LIN {X 0,Y 509.374,Z 538.173,A -85,B 0,C 180,E1 19045.4,E2 19045.4} C_VEL
LIN {X 0,Y 505.626,Z 523.597,A -85,B 0,C 180,E1 19044.365,E2 19044.365} C_VEL
LIN {X 0,Y 504.714,Z 520.545,A -85,B 0,C 180,E1 19044.099,E2 19044.099} C_VEL
LIN {X 0,Y 504.683,Z 520.186,A -85,B 0,C 180,E1 19043.675,E2 19043.675} C_VEL
LIN {X 0,Y 504.675,Z 520.134,A -85,B 0,C 180,E1 19040.214,E2 19040.214} C_VEL
LIN {X 0,Y 504.748,Z 520.47,A -85,B 0,C 180,E1 19039.175,E2 19039.175} C_VEL
LIN {X 0,Y 506.259,Z 524.019,A -85,B 0,C 180,E1 19038.577,E2 19038.577} C_VEL
LIN {X 0,Y 514.07,Z 540.46,A -85,B 0,C 180,E1 19036.024,E2 19036.024} C_VEL
LIN {X 0,Y 516.619,Z 546.048,A -85,B 0,C 180,E1 19035.262,E2 19035.262} C_VEL
LIN {X 0,Y 526.038,Z 560.599,A -85,B 0,C 180,E1 19034.052,E2 19034.052} C_VEL
LIN {X 0,Y 527.632,Z 568.688,A -85,B 0,C 180,E1 19033.753,E2 19033.753} C_VEL
LIN {X 0,Y 524.708,Z 775.867,A -85,B 0,C 180,E1 19030.439,E2 19030.439} C_VEL
LIN {X 0,Y 522.743,Z 892.473,A -85,B 0,C 180,E1 19028.548,E2 19028.548} C_VEL
LIN {X 0,Y 521.824,Z 915.213,A -85,B 0,C 180,E1 19027.996,E2 19027.996} C_VEL
LIN {X 0,Y 520.789,Z 935.158,A -85,B 0,C 180,E1 19027.346,E2 19027.346} C_VEL
LIN {X 0,Y 519.279,Z 958.378,A -85,B 0,C 180,E1 19026.374,E2 19026.374} C_VEL
LIN {X 0,Y 517.768,Z 979.695,A -85,B 0,C 180,E1 19025.268,E2 19025.268} C_VEL
LIN {X 0,Y 516.05,Z 1000.225,A -85,B 0,C 180,E1 19023.978,E2 19023.978} C_VEL
LIN {X 0,Y 514.336,Z 1020.252,A -85,B 0,C 180,E1 19022.508,E2 19022.508} C_VEL
LIN {X 0,Y 512.59,Z 1039.264,A -85,B 0,C 180,E1 19020.865,E2 19020.865} C_VEL
LIN {X 0,Y 510.801,Z 1058.785,A -85,B 0,C 180,E1 19018.914,E2 19018.914} C_VEL
LIN {X 0,Y 509.332,Z 1075.15,A -85,B 0,C 180,E1 19017.03,E2 19017.03} C_VEL
LIN {X 0,Y 507.958,Z 1091.142,A -85,B 0,C 180,E1 19014.913,E2 19014.913} C_VEL
LIN {X 0,Y 506.773,Z 1106.221,A -85,B 0,C 180,E1 19012.627,E2 19012.627} C_VEL
LIN {X 0,Y 505.853,Z 1119.088,A -85,B 0,C 180,E1 19010.358,E2 19010.358} C_VEL
LIN {X 0,Y 505.083,Z 1131.807,A -85,B 0,C 180,E1 19007.75,E2 19007.75} C_VEL
LIN {X 0,Y 504.598,Z 1141.528,A -85,B 0,C 180,E1 19005.398,E2 19005.398} C_VEL
LIN {X 0,Y 504.238,Z 1150.346,A -85,B 0,C 180,E1 19002.832,E2 19002.832} C_VEL
LIN {X 0,Y 504.07,Z 1156.866,A -85,B 0,C 180,E1 19000.515,E2 19000.515} C_VEL
LIN {X 0,Y 503.966,Z 1162.635,A -85,B 0,C 180,E1 18997.868,E2 18997.868} C_VEL
LIN {X 0,Y 503.904,Z 1166.278,A -85,B 0,C 180,E1 18995.58,E2 18995.58} C_VEL
LIN {X 0,Y 503.889,Z 1168.919,A -85,B 0,C 180,E1 18992.957,E2 18992.957} C_VEL
LIN {X 0,Y 503.884,Z 1169.872,A -85,B 0,C 180,E1 18990.682,E2 18990.682} C_VEL
LIN {X 0,Y 503.907,Z 1169.526,A -85,B 0,C 180,E1 18988.067,E2 18988.067} C_VEL
LIN {X 0,Y 503.913,Z 1167.729,A -85,B 0,C 180,E1 18985.676,E2 18985.676} C_VEL
LIN {X 0,Y 503.923,Z 1164.494,A -85,B 0,C 180,E1 18983.163,E2 18983.163} C_VEL
LIN {X 0,Y 504.003,Z 1159.828,A -85,B 0,C 180,E1 18980.753,E2 18980.753} C_VEL
LIN {X 0,Y 504.156,Z 1153.517,A -85,B 0,C 180,E1 18978.213,E2 18978.213} C_VEL
LIN {X 0,Y 504.423,Z 1145.344,A -85,B 0,C 180,E1 18975.654,E2 18975.654} C_VEL
LIN {X 0,Y 504.885,Z 1135.421,A -85,B 0,C 180,E1 18973.075,E2 18973.075} C_VEL
LIN {X 0,Y 505.497,Z 1124.573,A -85,B 0,C 180,E1 18970.712,E2 18970.712} C_VEL
LIN {X 0,Y 506.398,Z 1111.156,A -85,B 0,C 180,E1 18968.21,E2 18968.21} C_VEL
LIN {X 0,Y 507.492,Z 1097.01,A -85,B 0,C 180,E1 18965.931,E2 18965.931} C_VEL
LIN {X 0,Y 508.795,Z 1081.335,A -85,B 0,C 180,E1 18963.758,E2 18963.758} C_VEL
LIN {X 0,Y 510.309,Z 1064.33,A -85,B 0,C 180,E1 18961.696,E2 18961.696} C_VEL
LIN {X 0,Y 511.832,Z 1047.548,A -85,B 0,C 180,E1 18959.927,E2 18959.927} C_VEL
LIN {X 0,Y 513.655,Z 1027.52,A -85,B 0,C 180,E1 18958.096,E2 18958.096} C_VEL
LIN {X 0,Y 515.411,Z 1008.083,A -85,B 0,C 180,E1 18956.568,E2 18956.568} C_VEL
LIN {X 0,Y 517.065,Z 987.821,A -85,B 0,C 180,E1 18955.218,E2 18955.218} C_VEL
LIN {X 0,Y 518.718,Z 967.181,A -85,B 0,C 180,E1 18954.054,E2 18954.054} C_VEL
LIN {X 0,Y 520.087,Z 946.602,A -85,B 0,C 180,E1 18953.106,E2 18953.106} C_VEL
LIN {X 0,Y 521.311,Z 925.729,A -85,B 0,C 180,E1 18952.321,E2 18952.321} C_VEL
LIN {X 0,Y 522.324,Z 902.992,A -85,B 0,C 180,E1 18951.682,E2 18951.682} C_VEL
LIN {X 0,Y 523.077,Z 879.403,A -85,B 0,C 180,E1 18951.217,E2 18951.217} C_VEL
LIN {X 0,Y 525.528,Z 712.407,A -85,B 0,C 180,E1 18948.56,E2 18948.56} C_VEL
LIN {X 0,Y 527.601,Z 563.686,A -85,B 0,C 180,E1 18946.153,E2 18946.153} C_VEL
LIN {X 0,Y 526.674,Z 559.647,A -85,B 0,C 180,E1 18945.992,E2 18945.992} C_VEL
LIN {X 0,Y 516.407,Z 544.042,A -85,B 0,C 180,E1 18944.654,E2 18944.654} C_VEL
LIN {X 0,Y 508.668,Z 528.582,A -85,B 0,C 180,E1 18942.545,E2 18942.545} C_VEL
LIN {X 0,Y 506.242,Z 523.996,A -85,B 0,C 180,E1 18941.875,E2 18941.875} C_VEL
LIN {X 0,Y 504.741,Z 520.388,A -85,B 0,C 180,E1 18941.325,E2 18941.325} C_VEL
LIN {X 0,Y 504.697,Z 520.161,A -85,B 0,C 180,E1 18937.771,E2 18937.771} C_VEL
LIN {X 0,Y 504.694,Z 520.181,A -85,B 0,C 180,E1 18934.238,E2 18934.238} C_VEL
LIN {X 0,Y 504.711,Z 520.174,A -85,B 0,C 180,E1 18930.708,E2 18930.708} C_VEL
LIN {X 0,Y 504.695,Z 520.153,A -85,B 0,C 180,E1 18927.186,E2 18927.186} C_VEL
LIN {X 0,Y 504.695,Z 520.179,A -85,B 0,C 180,E1 18923.713,E2 18923.713} C_VEL
LIN {X 0,Y 504.703,Z 520.168,A -85,B 0,C 180,E1 18920.164,E2 18920.164} C_VEL
LIN {X 0,Y 504.697,Z 520.159,A -85,B 0,C 180,E1 18916.694,E2 18916.694} C_VEL
LIN {X 0,Y 504.694,Z 520.17,A -85,B 0,C 180,E1 18913.169,E2 18913.169} C_VEL
LIN {X 0,Y 504.699,Z 520.157,A -85,B 0,C 180,E1 18909.694,E2 18909.694} C_VEL
LIN {X 0,Y 504.697,Z 520.176,A -85,B 0,C 180,E1 18906.141,E2 18906.141} C_VEL
LIN {X 0,Y 504.695,Z 520.173,A -85,B 0,C 180,E1 18902.611,E2 18902.611} C_VEL
LIN {X 0,Y 504.702,Z 520.173,A -85,B 0,C 180,E1 18899.092,E2 18899.092} C_VEL
LIN {X 0,Y 504.695,Z 520.178,A -85,B 0,C 180,E1 18895.568,E2 18895.568} C_VEL
LIN {X 0,Y 504.698,Z 520.171,A -85,B 0,C 180,E1 18892.119,E2 18892.119} C_VEL
LIN {X 0,Y 504.695,Z 520.16,A -85,B 0,C 180,E1 18888.573,E2 18888.573} C_VEL
LIN {X 0,Y 504.693,Z 520.179,A -85,B 0,C 180,E1 18884.958,E2 18884.958} C_VEL
LIN {X 0,Y 504.698,Z 520.155,A -85,B 0,C 180,E1 18881.52,E2 18881.52} C_VEL
LIN {X 0,Y 504.698,Z 520.177,A -85,B 0,C 180,E1 18877.996,E2 18877.996} C_VEL
LIN {X 0,Y 504.69,Z 520.153,A -85,B 0,C 180,E1 18874.412,E2 18874.412} C_VEL
LIN {X 0,Y 504.701,Z 520.175,A -85,B 0,C 180,E1 18870.887,E2 18870.887} C_VEL
LIN {X 0,Y 504.7,Z 520.176,A -85,B 0,C 180,E1 18867.349,E2 18867.349} C_VEL
LIN {X 0,Y 504.685,Z 520.158,A -85,B 0,C 180,E1 18863.739,E2 18863.739} C_VEL
LIN {X 0,Y 504.699,Z 520.158,A -85,B 0,C 180,E1 18860.363,E2 18860.363} C_VEL
LIN {X 0,Y 504.689,Z 520.163,A -85,B 0,C 180,E1 18856.883,E2 18856.883} C_VEL
LIN {X 0,Y 504.772,Z 520.605,A -85,B 0,C 180,E1 18856.246,E2 18856.246} C_VEL
LIN {X 0,Y 506.506,Z 524.334,A -85,B 0,C 180,E1 18855.668,E2 18855.668} C_VEL
LIN {X 0,Y 515.146,Z 542.071,A -85,B 0,C 180,E1 18853.131,E2 18853.131} C_VEL
LIN {X 0,Y 516.768,Z 545.52,A -85,B 0,C 180,E1 18852.666,E2 18852.666} C_VEL
LIN {X 0,Y 517.661,Z 549.436,A -85,B 0,C 180,E1 18852.245,E2 18852.245} C_VEL
LIN {X 0,Y 517.414,Z 555.801,A -85,B 0,C 180,E1 18851.744,E2 18851.744} C_VEL
LIN {X 0,Y 513.944,Z 574.599,A -85,B 0,C 180,E1 18850.556,E2 18850.556} C_VEL
LIN {X 0,Y 513.868,Z 575.564,A -85,B 0,C 180,E1 18850.486,E2 18850.486} C_VEL
LIN {X 0,Y 513.159,Z 588.697,A -85,B 0,C 180,E1 18849.537,E2 18849.537} C_VEL
LIN {X 0,Y 516.897,Z 611.864,A -85,B 0,C 180,E1 18848.752,E2 18848.752} C_VEL
LIN {X 0,Y 513.011,Z 833.068,A -85,B 0,C 180,E1 18845.203,E2 18845.203} C_VEL
LIN {X 0,Y 511.794,Z 896.976,A -85,B 0,C 180,E1 18844.15,E2 18844.15} C_VEL
LIN {X 0,Y 510.861,Z 917.747,A -85,B 0,C 180,E1 18843.613,E2 18843.613} C_VEL
LIN {X 0,Y 509.667,Z 940.451,A -85,B 0,C 180,E1 18842.816,E2 18842.816} C_VEL
LIN {X 0,Y 508.463,Z 960.06,A -85,B 0,C 180,E1 18841.936,E2 18841.936} C_VEL
LIN {X 0,Y 506.93,Z 980.559,A -85,B 0,C 180,E1 18840.786,E2 18840.786} C_VEL
LIN {X 0,Y 505.393,Z 1000.249,A -85,B 0,C 180,E1 18839.448,E2 18839.448} C_VEL
LIN {X 0,Y 503.85,Z 1018.516,A -85,B 0,C 180,E1 18837.984,E2 18837.984} C_VEL
LIN {X 0,Y 502.296,Z 1036.377,A -85,B 0,C 180,E1 18836.289,E2 18836.289} C_VEL
LIN {X 0,Y 500.843,Z 1052.997,A -85,B 0,C 180,E1 18834.448,E2 18834.448} C_VEL
LIN {X 0,Y 499.563,Z 1068.367,A -85,B 0,C 180,E1 18832.475,E2 18832.475} C_VEL
LIN {X 0,Y 498.455,Z 1082.852,A -85,B 0,C 180,E1 18830.305,E2 18830.305} C_VEL
LIN {X 0,Y 497.584,Z 1095.279,A -85,B 0,C 180,E1 18828.11,E2 18828.11} C_VEL
LIN {X 0,Y 496.885,Z 1107.121,A -85,B 0,C 180,E1 18825.643,E2 18825.643} C_VEL
LIN {X 0,Y 496.443,Z 1116.603,A -85,B 0,C 180,E1 18823.274,E2 18823.274} C_VEL
LIN {X 0,Y 496.165,Z 1124.245,A -85,B 0,C 180,E1 18820.919,E2 18820.919} C_VEL
LIN {X 0,Y 496.006,Z 1130.548,A -85,B 0,C 180,E1 18818.462,E2 18818.462} C_VEL
LIN {X 0,Y 495.933,Z 1135.255,A -85,B 0,C 180,E1 18816.018,E2 18816.018} C_VEL
LIN {X 0,Y 495.907,Z 1138.243,A -85,B 0,C 180,E1 18813.583,E2 18813.583} C_VEL
LIN {X 0,Y 495.908,Z 1139.793,A -85,B 0,C 180,E1 18811.04,E2 18811.04} C_VEL
LIN {X 0,Y 495.908,Z 1139.767,A -85,B 0,C 180,E1 18808.729,E2 18808.729} C_VEL
LIN {X 0,Y 495.907,Z 1138.105,A -85,B 0,C 180,E1 18806.185,E2 18806.185} C_VEL
LIN {X 0,Y 495.941,Z 1134.893,A -85,B 0,C 180,E1 18803.685,E2 18803.685} C_VEL
LIN {X 0,Y 496.014,Z 1130.234,A -85,B 0,C 180,E1 18801.304,E2 18801.304} C_VEL
LIN {X 0,Y 496.175,Z 1123.81,A -85,B 0,C 180,E1 18798.846,E2 18798.846} C_VEL
LIN {X 0,Y 496.469,Z 1116.095,A -85,B 0,C 180,E1 18796.49,E2 18796.49} C_VEL
LIN {X 0,Y 496.927,Z 1106.429,A -85,B 0,C 180,E1 18794.108,E2 18794.108} C_VEL
LIN {X 0,Y 497.605,Z 1094.92,A -85,B 0,C 180,E1 18791.732,E2 18791.732} C_VEL
LIN {X 0,Y 498.501,Z 1082.19,A -85,B 0,C 180,E1 18789.501,E2 18789.501} C_VEL
LIN {X 0,Y 499.582,Z 1068.129,A -85,B 0,C 180,E1 18787.402,E2 18787.402} C_VEL
LIN {X 0,Y 500.879,Z 1052.572,A -85,B 0,C 180,E1 18785.411,E2 18785.411} C_VEL
LIN {X 0,Y 502.377,Z 1035.417,A -85,B 0,C 180,E1 18783.524,E2 18783.524} C_VEL
LIN {X 0,Y 503.893,Z 1018.046,A -85,B 0,C 180,E1 18781.883,E2 18781.883} C_VEL
LIN {X 0,Y 505.437,Z 999.747,A -85,B 0,C 180,E1 18780.425,E2 18780.425} C_VEL
LIN {X 0,Y 506.985,Z 979.853,A -85,B 0,C 180,E1 18779.081,E2 18779.081} C_VEL
LIN {X 0,Y 508.446,Z 960.379,A -85,B 0,C 180,E1 18777.99,E2 18777.99} C_VEL
LIN {X 0,Y 509.681,Z 940.217,A -85,B 0,C 180,E1 18777.084,E2 18777.084} C_VEL
LIN {X 0,Y 510.897,Z 917.075,A -85,B 0,C 180,E1 18776.277,E2 18776.277} C_VEL
LIN {X 0,Y 511.811,Z 896.306,A -85,B 0,C 180,E1 18775.746,E2 18775.746} C_VEL
LIN {X 0,Y 513.921,Z 783.082,A -85,B 0,C 180,E1 18773.904,E2 18773.904} C_VEL
LIN {X 0,Y 516.736,Z 613.605,A -85,B 0,C 180,E1 18771.173,E2 18771.173} C_VEL
LIN {X 0,Y 511.613,Z 588.579,A -85,B 0,C 180,E1 18770.179,E2 18770.179} C_VEL
LIN {X 0,Y 513.574,Z 559.712,A -85,B 0,C 180,E1 18767.55,E2 18767.55} C_VEL
LIN {X 0,Y 507.022,Z 544.118,A -85,B 0,C 180,E1 18765.229,E2 18765.229} C_VEL
LIN {X 0,Y 500.324,Z 529.196,A -85,B 0,C 180,E1 18762.802,E2 18762.802} C_VEL
LIN {X 0,Y 496.818,Z 521.605,A -85,B 0,C 180,E1 18761.462,E2 18761.462} C_VEL
LIN {X 0,Y 496.742,Z 521.125,A -85,B 0,C 180,E1 18760.814,E2 18760.814} C_VEL
LIN {X 0,Y 496.756,Z 521.438,A -85,B 0,C 180,E1 18758.385,E2 18758.385} C_VEL
LIN {X 0,Y 504.618,Z 543.801,A -85,B 0,C 180,E1 18755.961,E2 18755.961} C_VEL
LIN {X 0,Y 505.837,Z 548.641,A -85,B 0,C 180,E1 18755.474,E2 18755.474} C_VEL
LIN {X 0,Y 504.883,Z 590.98,A -85,B 0,C 180,E1 18752.048,E2 18752.048} C_VEL
LIN {X 0,Y 503.801,Z 630.683,A -85,B 0,C 180,E1 18748.834,E2 18748.834} C_VEL
LIN {X 0,Y 502.476,Z 673.939,A -85,B 0,C 180,E1 18745.33,E2 18745.33} C_VEL
LIN {X 0,Y 501.367,Z 709.763,A -85,B 0,C 180,E1 18742.454,E2 18742.454} C_VEL
LIN {X 0,Y 502.49,Z 720.165,A -85,B 0,C 180,E1 18742.24,E2 18742.24} C_VEL
LIN {X 0,Y 501.055,Z 879.658,A -85,B 0,C 180,E1 18739.834,E2 18739.834} C_VEL
LIN {X 0,Y 500.731,Z 897.059,A -85,B 0,C 180,E1 18739.361,E2 18739.361} C_VEL
LIN {X 0,Y 500.263,Z 913.355,A -85,B 0,C 180,E1 18738.705,E2 18738.705} C_VEL
LIN {X 0,Y 499.681,Z 929.581,A -85,B 0,C 180,E1 18737.828,E2 18737.828} C_VEL
LIN {X 0,Y 499.025,Z 944.8,A -85,B 0,C 180,E1 18736.77,E2 18736.77} C_VEL
LIN {X 0,Y 498.371,Z 958.85,A -85,B 0,C 180,E1 18735.536,E2 18735.536} C_VEL
LIN {X 0,Y 497.722,Z 971.827,A -85,B 0,C 180,E1 18734.128,E2 18734.128} C_VEL
LIN {X 0,Y 497.144,Z 983.648,A -85,B 0,C 180,E1 18732.546,E2 18732.546} C_VEL
LIN {X 0,Y 496.667,Z 994.101,A -85,B 0,C 180,E1 18730.791,E2 18730.791} C_VEL
LIN {X 0,Y 496.318,Z 1002.856,A -85,B 0,C 180,E1 18728.924,E2 18728.924} C_VEL
LIN {X 0,Y 496.099,Z 1009.578,A -85,B 0,C 180,E1 18727.062,E2 18727.062} C_VEL
LIN {X 0,Y 495.978,Z 1014.779,A -85,B 0,C 180,E1 18725.089,E2 18725.089} C_VEL
LIN {X 0,Y 495.929,Z 1018.358,A -85,B 0,C 180,E1 18723.005,E2 18723.005} C_VEL
LIN {X 0,Y 495.92,Z 1020.068,A -85,B 0,C 180,E1 18720.924,E2 18720.924} C_VEL
LIN {X 0,Y 495.924,Z 1020.017,A -85,B 0,C 180,E1 18718.845,E2 18718.845} C_VEL
LIN {X 0,Y 495.933,Z 1018.218,A -85,B 0,C 180,E1 18716.764,E2 18716.764} C_VEL
LIN {X 0,Y 495.996,Z 1014.584,A -85,B 0,C 180,E1 18714.68,E2 18714.68} C_VEL
LIN {X 0,Y 496.133,Z 1009.313,A -85,B 0,C 180,E1 18712.706,E2 18712.706} C_VEL
LIN {X 0,Y 496.402,Z 1002.018,A -85,B 0,C 180,E1 18710.727,E2 18710.727} C_VEL
LIN {X 0,Y 496.756,Z 993.678,A -85,B 0,C 180,E1 18708.977,E2 18708.977} C_VEL
LIN {X 0,Y 497.217,Z 983.868,A -85,B 0,C 180,E1 18707.339,E2 18707.339} C_VEL
LIN {X 0,Y 497.788,Z 972.555,A -85,B 0,C 180,E1 18705.816,E2 18705.816} C_VEL
LIN {X 0,Y 498.431,Z 959.663,A -85,B 0,C 180,E1 18704.407,E2 18704.407} C_VEL
LIN {X 0,Y 499.06,Z 945.596,A -85,B 0,C 180,E1 18703.172,E2 18703.172} C_VEL
LIN {X 0,Y 499.651,Z 931.225,A -85,B 0,C 180,E1 18702.172,E2 18702.172} C_VEL
LIN {X 0,Y 500.187,Z 914.88,A -85,B 0,C 180,E1 18701.287,E2 18701.287} C_VEL
LIN {X 0,Y 500.618,Z 898.01,A -85,B 0,C 180,E1 18700.615,E2 18700.615} C_VEL
LIN {X 0,Y 500.878,Z 880.613,A -85,B 0,C 180,E1 18700.159,E2 18700.159} C_VEL
LIN {X 0,Y 502.04,Z 716.903,A -85,B 0,C 180,E1 18697.709,E2 18697.709} C_VEL
LIN {X 0,Y 501.572,Z 712.774,A -85,B 0,C 180,E1 18697.589,E2 18697.589} C_VEL
LIN {X 0,Y 502.647,Z 670.001,A -85,B 0,C 180,E1 18694.238,E2 18694.238} C_VEL
LIN {X 0,Y 503.155,Z 631.96,A -85,B 0,C 180,E1 18691.386,E2 18691.386} C_VEL
LIN {X 0,Y 503.12,Z 597.05,A -85,B 0,C 180,E1 18688.889,E2 18688.889} C_VEL
LIN {X 0,Y 502.621,Z 562.387,A -85,B 0,C 180,E1 18686.563,E2 18686.563} C_VEL
LIN {X 0,Y 501.893,Z 540.312,A -85,B 0,C 180,E1 18685.163,E2 18685.163} C_VEL
LIN {X 0,Y 498.305,Z 526.321,A -85,B 0,C 180,E1 18684.158,E2 18684.158} C_VEL
LIN {X 0,Y 496.798,Z 521.567,A -85,B 0,C 180,E1 18683.756,E2 18683.756} C_VEL
LIN {X 0,Y 496.763,Z 521.172,A -85,B 0,C 180,E1 18683.426,E2 18683.426} C_VEL
LIN {X 0,Y 496.772,Z 521.367,A -85,B 0,C 180,E1 18680.153,E2 18680.153} C_VEL
LIN {X 0,Y 498.226,Z 524.831,A -85,B 0,C 180,E1 18679.517,E2 18679.517} C_VEL
LIN {X 0,Y 504.997,Z 538.88,A -85,B 0,C 180,E1 18677.226,E2 18677.226} C_VEL
LIN {X 0,Y 508.659,Z 546.653,A -85,B 0,C 180,E1 18676.082,E2 18676.082} C_VEL
LIN {X 0,Y 520.561,Z 564.965,A -85,B 0,C 180,E1 18674.505,E2 18674.505} C_VEL
LIN {X 0,Y 521.575,Z 570.604,A -85,B 0,C 180,E1 18674.302,E2 18674.302} C_VEL
LIN {X 0,Y 518.254,Z 778.338,A -85,B 0,C 180,E1 18670.928,E2 18670.928} C_VEL
LIN {X 0,Y 516.543,Z 889.73,A -85,B 0,C 180,E1 18669.155,E2 18669.155} C_VEL
LIN {X 0,Y 515.572,Z 913.827,A -85,B 0,C 180,E1 18668.588,E2 18668.588} C_VEL
LIN {X 0,Y 514.484,Z 933.42,A -85,B 0,C 180,E1 18667.954,E2 18667.954} C_VEL
LIN {X 0,Y 512.959,Z 955.807,A -85,B 0,C 180,E1 18667.035,E2 18667.035} C_VEL
LIN {X 0,Y 511.293,Z 977.07,A -85,B 0,C 180,E1 18665.944,E2 18665.944} C_VEL
LIN {X 0,Y 509.443,Z 998.326,A -85,B 0,C 180,E1 18664.624,E2 18664.624} C_VEL
LIN {X 0,Y 507.602,Z 1017.814,A -85,B 0,C 180,E1 18663.202,E2 18663.202} C_VEL
LIN {X 0,Y 505.712,Z 1037.012,A -85,B 0,C 180,E1 18661.555,E2 18661.555} C_VEL
LIN {X 0,Y 503.885,Z 1055.445,A -85,B 0,C 180,E1 18659.741,E2 18659.741} C_VEL
LIN {X 0,Y 502.167,Z 1072.616,A -85,B 0,C 180,E1 18657.77,E2 18657.77} C_VEL
LIN {X 0,Y 500.57,Z 1089.447,A -85,B 0,C 180,E1 18655.56,E2 18655.56} C_VEL
LIN {X 0,Y 499.284,Z 1103.97,A -85,B 0,C 180,E1 18653.36,E2 18653.36} C_VEL
LIN {X 0,Y 498.176,Z 1117.816,A -85,B 0,C 180,E1 18650.932,E2 18650.932} C_VEL
LIN {X 0,Y 497.354,Z 1129.723,A -85,B 0,C 180,E1 18648.52,E2 18648.52} C_VEL
LIN {X 0,Y 496.736,Z 1140.15,A -85,B 0,C 180,E1 18646.007,E2 18646.007} C_VEL
LIN {X 0,Y 496.322,Z 1149.441,A -85,B 0,C 180,E1 18643.342,E2 18643.342} C_VEL
LIN {X 0,Y 496.105,Z 1156.26,A -85,B 0,C 180,E1 18640.921,E2 18640.921} C_VEL
LIN {X 0,Y 495.971,Z 1162.428,A -85,B 0,C 180,E1 18638.113,E2 18638.113} C_VEL
LIN {X 0,Y 495.905,Z 1166.119,A -85,B 0,C 180,E1 18635.786,E2 18635.786} C_VEL
LIN {X 0,Y 495.885,Z 1168.85,A -85,B 0,C 180,E1 18633.121,E2 18633.121} C_VEL
LIN {X 0,Y 495.885,Z 1169.85,A -85,B 0,C 180,E1 18630.809,E2 18630.809} C_VEL
LIN {X 0,Y 495.904,Z 1169.658,A -85,B 0,C 180,E1 18628.267,E2 18628.267} C_VEL
LIN {X 0,Y 495.914,Z 1167.842,A -85,B 0,C 180,E1 18625.722,E2 18625.722} C_VEL
LIN {X 0,Y 495.925,Z 1164.681,A -85,B 0,C 180,E1 18623.168,E2 18623.168} C_VEL
LIN {X 0,Y 496.007,Z 1159.828,A -85,B 0,C 180,E1 18620.603,E2 18620.603} C_VEL
LIN {X 0,Y 496.185,Z 1153.517,A -85,B 0,C 180,E1 18618.021,E2 18618.021} C_VEL
LIN {X 0,Y 496.491,Z 1145.343,A -85,B 0,C 180,E1 18615.42,E2 18615.42} C_VEL
LIN {X 0,Y 497.005,Z 1135.42,A -85,B 0,C 180,E1 18612.799,E2 18612.799} C_VEL
LIN {X 0,Y 497.691,Z 1124.575,A -85,B 0,C 180,E1 18610.397,E2 18610.397} C_VEL
LIN {X 0,Y 498.691,Z 1111.154,A -85,B 0,C 180,E1 18607.856,E2 18607.856} C_VEL
LIN {X 0,Y 499.892,Z 1097.012,A -85,B 0,C 180,E1 18605.542,E2 18605.542} C_VEL
LIN {X 0,Y 501.338,Z 1081.159,A -85,B 0,C 180,E1 18603.313,E2 18603.313} C_VEL
LIN {X 0,Y 503.041,Z 1063.833,A -85,B 0,C 180,E1 18601.19,E2 18601.19} C_VEL
LIN {X 0,Y 504.708,Z 1046.955,A -85,B 0,C 180,E1 18599.394,E2 18599.394} C_VEL
LIN {X 0,Y 506.661,Z 1027.449,A -85,B 0,C 180,E1 18597.596,E2 18597.596} C_VEL
LIN {X 0,Y 508.468,Z 1008.89,A -85,B 0,C 180,E1 18596.118,E2 18596.118} C_VEL
LIN {X 0,Y 510.36,Z 987.818,A -85,B 0,C 180,E1 18594.694,E2 18594.694} C_VEL
LIN {X 0,Y 512.135,Z 967.281,A -85,B 0,C 180,E1 18593.524,E2 18593.524} C_VEL
LIN {X 0,Y 513.653,Z 946.07,A -85,B 0,C 180,E1 18592.54,E2 18592.54} C_VEL
LIN {X 0,Y 515.046,Z 924.001,A -85,B 0,C 180,E1 18591.712,E2 18591.712} C_VEL
LIN {X 0,Y 516.102,Z 901.806,A -85,B 0,C 180,E1 18591.102,E2 18591.102} C_VEL
LIN {X 0,Y 516.881,Z 877.187,A -85,B 0,C 180,E1 18590.625,E2 18590.625} C_VEL
LIN {X 0,Y 519.937,Z 666.947,A -85,B 0,C 180,E1 18587.287,E2 18587.287} C_VEL
LIN {X 0,Y 521.512,Z 565.132,A -85,B 0,C 180,E1 18585.592,E2 18585.592} C_VEL
LIN {X 0,Y 520.827,Z 563.461,A -85,B 0,C 180,E1 18585.494,E2 18585.494} C_VEL
LIN {X 0,Y 508.356,Z 544.574,A -85,B 0,C 180,E1 18583.814,E2 18583.814} C_VEL
LIN {X 0,Y 500.859,Z 529.715,A -85,B 0,C 180,E1 18581.702,E2 18581.702} C_VEL
LIN {X 0,Y 498.39,Z 525.082,A -85,B 0,C 180,E1 18580.996,E2 18580.996} C_VEL
LIN {X 0,Y 496.805,Z 521.468,A -85,B 0,C 180,E1 18580.435,E2 18580.435} C_VEL
LIN {X 0,Y 496.773,Z 521.163,A -85,B 0,C 180,E1 18579.197,E2 18579.197} C_VEL
LIN {X 0,Y 496.758,Z 521.155,A -85,B 0,C 180,E1 18575.569,E2 18575.569} C_VEL
LIN {X 0,Y 496.753,Z 521.141,A -85,B 0,C 180,E1 18572.071,E2 18572.071} C_VEL
LIN {X 0,Y 496.767,Z 521.152,A -85,B 0,C 180,E1 18568.49,E2 18568.49} C_VEL
LIN {X 0,Y 496.758,Z 521.17,A -85,B 0,C 180,E1 18564.876,E2 18564.876} C_VEL
LIN {X 0,Y 496.759,Z 521.137,A -85,B 0,C 180,E1 18561.365,E2 18561.365} C_VEL
LIN {X 0,Y 496.763,Z 521.165,A -85,B 0,C 180,E1 18557.814,E2 18557.814} C_VEL
LIN {X 0,Y 496.75,Z 521.143,A -85,B 0,C 180,E1 18554.334,E2 18554.334} C_VEL
LIN {X 0,Y 496.763,Z 521.158,A -85,B 0,C 180,E1 18550.788,E2 18550.788} C_VEL
LIN {X 0,Y 496.76,Z 521.148,A -85,B 0,C 180,E1 18547.168,E2 18547.168} C_VEL
LIN {X 0,Y 496.751,Z 521.159,A -85,B 0,C 180,E1 18543.693,E2 18543.693} C_VEL
LIN {X 0,Y 496.771,Z 521.162,A -85,B 0,C 180,E1 18540.115,E2 18540.115} C_VEL
LIN {X 0,Y 496.761,Z 521.163,A -85,B 0,C 180,E1 18536.538,E2 18536.538} C_VEL
LIN {X 0,Y 496.75,Z 521.159,A -85,B 0,C 180,E1 18533.063,E2 18533.063} C_VEL
LIN {X 0,Y 496.765,Z 521.158,A -85,B 0,C 180,E1 18529.563,E2 18529.563} C_VEL
LIN {X 0,Y 496.761,Z 521.149,A -85,B 0,C 180,E1 18525.966,E2 18525.966} C_VEL
LIN {X 0,Y 496.749,Z 521.156,A -85,B 0,C 180,E1 18522.427,E2 18522.427} C_VEL
LIN {X 0,Y 496.765,Z 521.156,A -85,B 0,C 180,E1 18518.882,E2 18518.882} C_VEL
LIN {X 0,Y 496.762,Z 521.143,A -85,B 0,C 180,E1 18515.377,E2 18515.377} C_VEL
LIN {X 0,Y 496.752,Z 521.169,A -85,B 0,C 180,E1 18511.837,E2 18511.837} C_VEL
LIN {X 0,Y 496.762,Z 521.143,A -85,B 0,C 180,E1 18508.309,E2 18508.309} C_VEL
LIN {X 0,Y 496.763,Z 521.145,A -85,B 0,C 180,E1 18504.803,E2 18504.803} C_VEL
LIN {X 0,Y 496.748,Z 521.163,A -85,B 0,C 180,E1 18501.245,E2 18501.245} C_VEL
LIN {X 0,Y 496.756,Z 521.167,A -85,B 0,C 180,E1 18497.62,E2 18497.62} C_VEL
LIN {X 0,Y 496.82,Z 521.646,A -85,B 0,C 180,E1 18497.151,E2 18497.151} C_VEL
LIN {X 0,Y 498.188,Z 524.802,A -85,B 0,C 180,E1 18496.655,E2 18496.655} C_VEL
LIN {X 0,Y 499.412,Z 527.156,A -85,B 0,C 180,E1 18496.282,E2 18496.282} C_VEL
LIN {X 0,Y 507.139,Z 542.59,A -85,B 0,C 180,E1 18493.976,E2 18493.976} C_VEL
LIN {X 0,Y 514.912,Z 559.739,A -85,B 0,C 180,E1 18491.677,E2 18491.677} C_VEL
LIN {X 0,Y 513.868,Z 575.564,A -85,B 0,C 180,E1 18490.486,E2 18490.486} C_VEL
LIN {X 0,Y 512.884,Z 580.226,A -85,B 0,C 180,E1 18490.235,E2 18490.235} C_VEL
LIN {X 0,Y 509.389,Z 590.178,A -85,B 0,C 180,E1 18490.016,E2 18490.016} C_VEL
LIN {X 0,Y 508.425,Z 596.069,A -85,B 0,C 180,E1 18489.899,E2 18489.899} C_VEL
LIN {X 0,Y 508.597,Z 598.238,A -85,B 0,C 180,E1 18489.831,E2 18489.831} C_VEL
LIN {X 0,Y 510.875,Z 613.611,A -85,B 0,C 180,E1 18489.32,E2 18489.32} C_VEL
LIN {X 0,Y 506.742,Z 838.077,A -85,B 0,C 180,E1 18485.698,E2 18485.698} C_VEL
LIN {X 0,Y 505.528,Z 897.301,A -85,B 0,C 180,E1 18484.711,E2 18484.711} C_VEL
LIN {X 0,Y 504.54,Z 917.913,A -85,B 0,C 180,E1 18484.173,E2 18484.173} C_VEL
LIN {X 0,Y 503.294,Z 938.408,A -85,B 0,C 180,E1 18483.448,E2 18483.448} C_VEL
LIN {X 0,Y 501.844,Z 958.154,A -85,B 0,C 180,E1 18482.544,E2 18482.544} C_VEL
LIN {X 0,Y 499.955,Z 980.569,A -85,B 0,C 180,E1 18481.264,E2 18481.264} C_VEL
LIN {X 0,Y 498.281,Z 1000.336,A -85,B 0,C 180,E1 18479.904,E2 18479.904} C_VEL
LIN {X 0,Y 496.625,Z 1018.459,A -85,B 0,C 180,E1 18478.434,E2 18478.434} C_VEL
LIN {X 0,Y 494.938,Z 1036.322,A -85,B 0,C 180,E1 18476.717,E2 18476.717} C_VEL
LIN {X 0,Y 493.36,Z 1052.809,A -85,B 0,C 180,E1 18474.868,E2 18474.868} C_VEL
LIN {X 0,Y 491.948,Z 1068.374,A -85,B 0,C 180,E1 18472.843,E2 18472.843} C_VEL
LIN {X 0,Y 490.73,Z 1082.855,A -85,B 0,C 180,E1 18470.64,E2 18470.64} C_VEL
LIN {X 0,Y 489.783,Z 1095.085,A -85,B 0,C 180,E1 18468.447,E2 18468.447} C_VEL
LIN {X 0,Y 489.028,Z 1106.608,A -85,B 0,C 180,E1 18466.023,E2 18466.023} C_VEL
LIN {X 0,Y 488.526,Z 1116.198,A -85,B 0,C 180,E1 18463.613,E2 18463.613} C_VEL
LIN {X 0,Y 488.201,Z 1124.005,A -85,B 0,C 180,E1 18461.182,E2 18461.182} C_VEL
LIN {X 0,Y 488.019,Z 1130.549,A -85,B 0,C 180,E1 18458.602,E2 18458.602} C_VEL
LIN {X 0,Y 487.937,Z 1135.256,A -85,B 0,C 180,E1 18456.117,E2 18456.117} C_VEL
LIN {X 0,Y 487.907,Z 1138.263,A -85,B 0,C 180,E1 18453.622,E2 18453.622} C_VEL
LIN {X 0,Y 487.908,Z 1139.793,A -85,B 0,C 180,E1 18451.057,E2 18451.057} C_VEL
LIN {X 0,Y 487.908,Z 1139.766,A -85,B 0,C 180,E1 18448.708,E2 18448.708} C_VEL
LIN {X 0,Y 487.907,Z 1138.218,A -85,B 0,C 180,E1 18446.24,E2 18446.24} C_VEL
LIN {X 0,Y 487.941,Z 1135.211,A -85,B 0,C 180,E1 18443.765,E2 18443.765} C_VEL
LIN {X 0,Y 488.02,Z 1130.487,A -85,B 0,C 180,E1 18441.28,E2 18441.28} C_VEL
LIN {X 0,Y 488.205,Z 1123.807,A -85,B 0,C 180,E1 18438.661,E2 18438.661} C_VEL
LIN {X 0,Y 488.53,Z 1116.092,A -85,B 0,C 180,E1 18436.266,E2 18436.266} C_VEL
LIN {X 0,Y 489.036,Z 1106.473,A -85,B 0,C 180,E1 18433.855,E2 18433.855} C_VEL
LIN {X 0,Y 489.792,Z 1094.915,A -85,B 0,C 180,E1 18431.43,E2 18431.43} C_VEL
LIN {X 0,Y 490.748,Z 1082.642,A -85,B 0,C 180,E1 18429.236,E2 18429.236} C_VEL
LIN {X 0,Y 491.972,Z 1068.125,A -85,B 0,C 180,E1 18427.032,E2 18427.032} C_VEL
LIN {X 0,Y 493.387,Z 1052.509,A -85,B 0,C 180,E1 18425.005,E2 18425.005} C_VEL
LIN {X 0,Y 495.019,Z 1035.407,A -85,B 0,C 180,E1 18423.099,E2 18423.099} C_VEL
LIN {X 0,Y 496.67,Z 1018.036,A -85,B 0,C 180,E1 18421.437,E2 18421.437} C_VEL
LIN {X 0,Y 498.336,Z 999.734,A -85,B 0,C 180,E1 18419.96,E2 18419.96} C_VEL
LIN {X 0,Y 500.012,Z 979.912,A -85,B 0,C 180,E1 18418.606,E2 18418.606} C_VEL
LIN {X 0,Y 501.821,Z 958.57,A -85,B 0,C 180,E1 18417.387,E2 18417.387} C_VEL
LIN {X 0,Y 503.276,Z 938.697,A -85,B 0,C 180,E1 18416.475,E2 18416.475} C_VEL
LIN {X 0,Y 504.563,Z 917.528,A -85,B 0,C 180,E1 18415.725,E2 18415.725} C_VEL
LIN {X 0,Y 505.545,Z 896.839,A -85,B 0,C 180,E1 18415.189,E2 18415.189} C_VEL
LIN {X 0,Y 507.233,Z 812.873,A -85,B 0,C 180,E1 18413.805,E2 18413.805} C_VEL
LIN {X 0,Y 510.741,Z 615.457,A -85,B 0,C 180,E1 18410.61,E2 18410.61} C_VEL
LIN {X 0,Y 505.153,Z 588.344,A -85,B 0,C 180,E1 18409.517,E2 18409.517} C_VEL
LIN {X 0,Y 506.989,Z 563.56,A -85,B 0,C 180,E1 18407.24,E2 18407.24} C_VEL
LIN {X 0,Y 499.687,Z 546.036,A -85,B 0,C 180,E1 18404.574,E2 18404.574} C_VEL
LIN {X 0,Y 493.717,Z 533.224,A -85,B 0,C 180,E1 18402.406,E2 18402.406} C_VEL
LIN {X 0,Y 490.181,Z 525.671,A -85,B 0,C 180,E1 18401.057,E2 18401.057} C_VEL
LIN {X 0,Y 488.811,Z 522.393,A -85,B 0,C 180,E1 18400.423,E2 18400.423} C_VEL
LIN {X 0,Y 488.848,Z 522.288,A -85,B 0,C 180,E1 18398.944,E2 18398.944} C_VEL
LIN {X 0,Y 489.264,Z 524.003,A -85,B 0,C 180,E1 18398.679,E2 18398.679} C_VEL
LIN {X 0,Y 496.707,Z 544.646,A -85,B 0,C 180,E1 18396.429,E2 18396.429} C_VEL
LIN {X 0,Y 498.628,Z 551.007,A -85,B 0,C 180,E1 18395.769,E2 18395.769} C_VEL
LIN {X 0,Y 497.567,Z 593.401,A -85,B 0,C 180,E1 18392.312,E2 18392.312} C_VEL
LIN {X 0,Y 496.46,Z 632.014,A -85,B 0,C 180,E1 18389.169,E2 18389.169} C_VEL
LIN {X 0,Y 495.078,Z 674.907,A -85,B 0,C 180,E1 18385.671,E2 18385.671} C_VEL
LIN {X 0,Y 493.936,Z 710.913,A -85,B 0,C 180,E1 18382.771,E2 18382.771} C_VEL
LIN {X 0,Y 495.01,Z 721.17,A -85,B 0,C 180,E1 18382.554,E2 18382.554} C_VEL
LIN {X 0,Y 493.425,Z 881.029,A -85,B 0,C 180,E1 18380.092,E2 18380.092} C_VEL
LIN {X 0,Y 493.096,Z 898.405,A -85,B 0,C 180,E1 18379.609,E2 18379.609} C_VEL
LIN {X 0,Y 492.579,Z 915.607,A -85,B 0,C 180,E1 18378.897,E2 18378.897} C_VEL
LIN {X 0,Y 491.979,Z 931.828,A -85,B 0,C 180,E1 18377.994,E2 18377.994} C_VEL
LIN {X 0,Y 491.295,Z 946.831,A -85,B 0,C 180,E1 18376.92,E2 18376.92} C_VEL
LIN {X 0,Y 490.615,Z 960.713,A -85,B 0,C 180,E1 18375.67,E2 18375.67} C_VEL
LIN {X 0,Y 489.933,Z 973.829,A -85,B 0,C 180,E1 18374.213,E2 18374.213} C_VEL
LIN {X 0,Y 489.339,Z 985.405,A -85,B 0,C 180,E1 18372.629,E2 18372.629} C_VEL
LIN {X 0,Y 488.863,Z 995.166,A -85,B 0,C 180,E1 18370.965,E2 18370.965} C_VEL
LIN {X 0,Y 488.485,Z 1004.011,A -85,B 0,C 180,E1 18369.068,E2 18369.068} C_VEL
LIN {X 0,Y 488.247,Z 1010.832,A -85,B 0,C 180,E1 18367.176,E2 18367.176} C_VEL
LIN {X 0,Y 488.109,Z 1016.081,A -85,B 0,C 180,E1 18365.171,E2 18365.171} C_VEL
LIN {X 0,Y 488.052,Z 1019.703,A -85,B 0,C 180,E1 18363.054,E2 18363.054} C_VEL
LIN {X 0,Y 488.047,Z 1021.485,A -85,B 0,C 180,E1 18360.939,E2 18360.939} C_VEL
LIN {X 0,Y 488.057,Z 1021.46,A -85,B 0,C 180,E1 18358.826,E2 18358.826} C_VEL
LIN {X 0,Y 488.074,Z 1019.655,A -85,B 0,C 180,E1 18356.712,E2 18356.712} C_VEL
LIN {X 0,Y 488.157,Z 1016.031,A -85,B 0,C 180,E1 18354.594,E2 18354.594} C_VEL
LIN {X 0,Y 488.311,Z 1010.708,A -85,B 0,C 180,E1 18352.589,E2 18352.589} C_VEL
LIN {X 0,Y 488.616,Z 1003.386,A -85,B 0,C 180,E1 18350.578,E2 18350.578} C_VEL
LIN {X 0,Y 489.002,Z 994.994,A -85,B 0,C 180,E1 18348.8,E2 18348.8} C_VEL
LIN {X 0,Y 489.495,Z 985.076,A -85,B 0,C 180,E1 18347.136,E2 18347.136} C_VEL
LIN {X 0,Y 490.1,Z 973.648,A -85,B 0,C 180,E1 18345.588,E2 18345.588} C_VEL
LIN {X 0,Y 490.774,Z 960.603,A -85,B 0,C 180,E1 18344.158,E2 18344.158} C_VEL
LIN {X 0,Y 491.388,Z 947.033,A -85,B 0,C 180,E1 18342.962,E2 18342.962} C_VEL
LIN {X 0,Y 491.991,Z 932.54,A -85,B 0,C 180,E1 18341.946,E2 18341.946} C_VEL
LIN {X 0,Y 492.532,Z 916.017,A -85,B 0,C 180,E1 18341.047,E2 18341.047} C_VEL
LIN {X 0,Y 492.948,Z 899.094,A -85,B 0,C 180,E1 18340.374,E2 18340.374} C_VEL
LIN {X 0,Y 493.188,Z 881.513,A -85,B 0,C 180,E1 18339.917,E2 18339.917} C_VEL
LIN {X 0,Y 494.544,Z 718.135,A -85,B 0,C 180,E1 18337.419,E2 18337.419} C_VEL
LIN {X 0,Y 494.193,Z 714.717,A -85,B 0,C 180,E1 18337.308,E2 18337.308} C_VEL
LIN {X 0,Y 495.179,Z 676.745,A -85,B 0,C 180,E1 18334.335,E2 18334.335} C_VEL
LIN {X 0,Y 495.731,Z 638.472,A -85,B 0,C 180,E1 18331.445,E2 18331.445} C_VEL
LIN {X 0,Y 495.758,Z 602.349,A -85,B 0,C 180,E1 18328.848,E2 18328.848} C_VEL
LIN {X 0,Y 495.277,Z 568.433,A -85,B 0,C 180,E1 18326.556,E2 18326.556} C_VEL
LIN {X 0,Y 494.435,Z 542.294,A -85,B 0,C 180,E1 18324.884,E2 18324.884} C_VEL
LIN {X 0,Y 491.097,Z 529.215,A -85,B 0,C 180,E1 18323.929,E2 18323.929} C_VEL
LIN {X 0,Y 488.889,Z 522.571,A -85,B 0,C 180,E1 18323.368,E2 18323.368} C_VEL
LIN {X 0,Y 488.831,Z 522.16,A -85,B 0,C 180,E1 18323.034,E2 18323.034} C_VEL
LIN {X 0,Y 488.866,Z 522.389,A -85,B 0,C 180,E1 18321.106,E2 18321.106} C_VEL
LIN {X 0,Y 490.247,Z 525.79,A -85,B 0,C 180,E1 18320.482,E2 18320.482} C_VEL
LIN {X 0,Y 495.349,Z 536.113,A -85,B 0,C 180,E1 18318.697,E2 18318.697} C_VEL
LIN {X 0,Y 500.753,Z 547.32,A -85,B 0,C 180,E1 18316.932,E2 18316.932} C_VEL
LIN {X 0,Y 515.106,Z 569.301,A -85,B 0,C 180,E1 18314.97,E2 18314.97} C_VEL
LIN {X 0,Y 515.56,Z 572.794,A -85,B 0,C 180,E1 18314.858,E2 18314.858} C_VEL
LIN {X 0,Y 511.929,Z 774.422,A -85,B 0,C 180,E1 18311.531,E2 18311.531} C_VEL
LIN {X 0,Y 509.973,Z 893.033,A -85,B 0,C 180,E1 18309.619,E2 18309.619} C_VEL
LIN {X 0,Y 509.009,Z 915.761,A -85,B 0,C 180,E1 18309.068,E2 18309.068} C_VEL
LIN {X 0,Y 507.873,Z 937.021,A -85,B 0,C 180,E1 18308.379,E2 18308.379} C_VEL
LIN {X 0,Y 506.272,Z 958.372,A -85,B 0,C 180,E1 18307.466,E2 18307.466} C_VEL
LIN {X 0,Y 504.496,Z 979.702,A -85,B 0,C 180,E1 18306.341,E2 18306.341} C_VEL
LIN {X 0,Y 502.523,Z 1000.123,A -85,B 0,C 180,E1 18305.031,E2 18305.031} C_VEL
LIN {X 0,Y 500.477,Z 1020.173,A -85,B 0,C 180,E1 18303.532,E2 18303.532} C_VEL
LIN {X 0,Y 498.425,Z 1039.259,A -85,B 0,C 180,E1 18301.843,E2 18301.843} C_VEL
LIN {X 0,Y 496.283,Z 1058.782,A -85,B 0,C 180,E1 18299.844,E2 18299.844} C_VEL
LIN {X 0,Y 494.578,Z 1074.89,A -85,B 0,C 180,E1 18297.939,E2 18297.939} C_VEL
LIN {X 0,Y 492.882,Z 1091.139,A -85,B 0,C 180,E1 18295.729,E2 18295.729} C_VEL
LIN {X 0,Y 491.447,Z 1106.225,A -85,B 0,C 180,E1 18293.374,E2 18293.374} C_VEL
LIN {X 0,Y 490.323,Z 1119.084,A -85,B 0,C 180,E1 18291.033,E2 18291.033} C_VEL
LIN {X 0,Y 489.408,Z 1131.288,A -85,B 0,C 180,E1 18288.461,E2 18288.461} C_VEL
LIN {X 0,Y 488.785,Z 1141.066,A -85,B 0,C 180,E1 18286.031,E2 18286.031} C_VEL
LIN {X 0,Y 488.333,Z 1150.348,A -85,B 0,C 180,E1 18283.257,E2 18283.257} C_VEL
LIN {X 0,Y 488.107,Z 1157.168,A -85,B 0,C 180,E1 18280.743,E2 18280.743} C_VEL
LIN {X 0,Y 487.975,Z 1162.635,A -85,B 0,C 180,E1 18278.128,E2 18278.128} C_VEL
LIN {X 0,Y 487.906,Z 1166.437,A -85,B 0,C 180,E1 18275.645,E2 18275.645} C_VEL
LIN {X 0,Y 487.89,Z 1168.986,A -85,B 0,C 180,E1 18272.937,E2 18272.937} C_VEL
LIN {X 0,Y 487.884,Z 1169.895,A -85,B 0,C 180,E1 18270.587,E2 18270.587} C_VEL
LIN {X 0,Y 487.914,Z 1169.392,A -85,B 0,C 180,E1 18267.769,E2 18267.769} C_VEL
LIN {X 0,Y 487.909,Z 1167.501,A -85,B 0,C 180,E1 18265.298,E2 18265.298} C_VEL
LIN {X 0,Y 487.932,Z 1163.874,A -85,B 0,C 180,E1 18262.583,E2 18262.583} C_VEL
LIN {X 0,Y 488.014,Z 1159.573,A -85,B 0,C 180,E1 18260.328,E2 18260.328} C_VEL
LIN {X 0,Y 488.213,Z 1153.517,A -85,B 0,C 180,E1 18257.822,E2 18257.822} C_VEL
LIN {X 0,Y 488.561,Z 1145.342,A -85,B 0,C 180,E1 18255.178,E2 18255.178} C_VEL
LIN {X 0,Y 489.13,Z 1135.419,A -85,B 0,C 180,E1 18252.513,E2 18252.513} C_VEL
LIN {X 0,Y 489.891,Z 1124.577,A -85,B 0,C 180,E1 18250.072,E2 18250.072} C_VEL
LIN {X 0,Y 490.992,Z 1111.152,A -85,B 0,C 180,E1 18247.49,E2 18247.49} C_VEL
LIN {X 0,Y 492.317,Z 1097.013,A -85,B 0,C 180,E1 18245.14,E2 18245.14} C_VEL
LIN {X 0,Y 493.87,Z 1081.332,A -85,B 0,C 180,E1 18242.901,E2 18242.901} C_VEL
LIN {X 0,Y 495.762,Z 1063.777,A -85,B 0,C 180,E1 18240.72,E2 18240.72} C_VEL
LIN {X 0,Y 497.616,Z 1046.55,A -85,B 0,C 180,E1 18238.865,E2 18238.865} C_VEL
LIN {X 0,Y 499.764,Z 1026.779,A -85,B 0,C 180,E1 18237.031,E2 18237.031} C_VEL
LIN {X 0,Y 501.82,Z 1007.265,A -85,B 0,C 180,E1 18235.469,E2 18235.469} C_VEL
LIN {X 0,Y 503.804,Z 986.808,A -85,B 0,C 180,E1 18234.094,E2 18234.094} C_VEL
LIN {X 0,Y 505.707,Z 966.078,A -85,B 0,C 180,E1 18232.913,E2 18232.913} C_VEL
LIN {X 0,Y 507.29,Z 945.161,A -85,B 0,C 180,E1 18231.944,E2 18231.944} C_VEL
LIN {X 0,Y 508.628,Z 923.534,A -85,B 0,C 180,E1 18231.156,E2 18231.156} C_VEL
LIN {X 0,Y 509.639,Z 901.371,A -85,B 0,C 180,E1 18230.563,E2 18230.563} C_VEL
LIN {X 0,Y 510.381,Z 875.527,A -85,B 0,C 180,E1 18230.078,E2 18230.078} C_VEL
LIN {X 0,Y 513.683,Z 671.929,A -85,B 0,C 180,E1 18226.798,E2 18226.798} C_VEL
LIN {X 0,Y 515.486,Z 568.099,A -85,B 0,C 180,E1 18225.05,E2 18225.05} C_VEL
LIN {X 0,Y 500.595,Z 545.629,A -85,B 0,C 180,E1 18223.007,E2 18223.007} C_VEL
LIN {X 0,Y 492.903,Z 530.633,A -85,B 0,C 180,E1 18220.781,E2 18220.781} C_VEL
LIN {X 0,Y 490.607,Z 526.252,A -85,B 0,C 180,E1 18220.091,E2 18220.091} C_VEL
LIN {X 0,Y 488.908,Z 522.688,A -85,B 0,C 180,E1 18219.515,E2 18219.515} C_VEL
LIN {X 0,Y 488.833,Z 522.154,A -85,B 0,C 180,E1 18219.176,E2 18219.176} C_VEL
LIN {X 0,Y 488.819,Z 522.143,A -85,B 0,C 180,E1 18215.502,E2 18215.502} C_VEL
LIN {X 0,Y 488.82,Z 522.128,A -85,B 0,C 180,E1 18211.911,E2 18211.911} C_VEL
LIN {X 0,Y 488.82,Z 522.136,A -85,B 0,C 180,E1 18208.329,E2 18208.329} C_VEL
LIN {X 0,Y 488.821,Z 522.158,A -85,B 0,C 180,E1 18204.744,E2 18204.744} C_VEL
LIN {X 0,Y 488.824,Z 522.125,A -85,B 0,C 180,E1 18201.1,E2 18201.1} C_VEL
LIN {X 0,Y 488.817,Z 522.152,A -85,B 0,C 180,E1 18197.498,E2 18197.498} C_VEL
LIN {X 0,Y 488.822,Z 522.136,A -85,B 0,C 180,E1 18193.967,E2 18193.967} C_VEL
LIN {X 0,Y 488.816,Z 522.138,A -85,B 0,C 180,E1 18190.303,E2 18190.303} C_VEL
LIN {X 0,Y 488.819,Z 522.141,A -85,B 0,C 180,E1 18186.695,E2 18186.695} C_VEL
LIN {X 0,Y 488.824,Z 522.146,A -85,B 0,C 180,E1 18183.048,E2 18183.048} C_VEL
LIN {X 0,Y 488.813,Z 522.152,A -85,B 0,C 180,E1 18179.531,E2 18179.531} C_VEL
LIN {X 0,Y 488.823,Z 522.15,A -85,B 0,C 180,E1 18176.012,E2 18176.012} C_VEL
LIN {X 0,Y 488.824,Z 522.146,A -85,B 0,C 180,E1 18172.359,E2 18172.359} C_VEL
LIN {X 0,Y 488.811,Z 522.138,A -85,B 0,C 180,E1 18168.795,E2 18168.795} C_VEL
LIN {X 0,Y 488.825,Z 522.147,A -85,B 0,C 180,E1 18165.186,E2 18165.186} C_VEL
LIN {X 0,Y 488.821,Z 522.129,A -85,B 0,C 180,E1 18161.639,E2 18161.639} C_VEL
LIN {X 0,Y 488.814,Z 522.157,A -85,B 0,C 180,E1 18158.144,E2 18158.144} C_VEL
LIN {X 0,Y 488.818,Z 522.125,A -85,B 0,C 180,E1 18154.561,E2 18154.561} C_VEL
LIN {X 0,Y 488.825,Z 522.153,A -85,B 0,C 180,E1 18151.002,E2 18151.002} C_VEL
LIN {X 0,Y 488.818,Z 522.15,A -85,B 0,C 180,E1 18147.43,E2 18147.43} C_VEL
LIN {X 0,Y 488.808,Z 522.131,A -85,B 0,C 180,E1 18143.761,E2 18143.761} C_VEL
LIN {X 0,Y 488.822,Z 522.13,A -85,B 0,C 180,E1 18140.272,E2 18140.272} C_VEL
LIN {X 0,Y 488.867,Z 522.441,A -85,B 0,C 180,E1 18138.161,E2 18138.161} C_VEL
LIN {X 0,Y 490.383,Z 526.015,A -85,B 0,C 180,E1 18137.554,E2 18137.554} C_VEL
LIN {X 0,Y 495.715,Z 536.348,A -85,B 0,C 180,E1 18135.894,E2 18135.894} C_VEL
LIN {X 0,Y 503.84,Z 553.238,A -85,B 0,C 180,E1 18133.421,E2 18133.421} C_VEL
LIN {X 0,Y 508.425,Z 563.733,A -85,B 0,C 180,E1 18132.023,E2 18132.023} C_VEL
LIN {X 0,Y 506.823,Z 588.14,A -85,B 0,C 180,E1 18130.202,E2 18130.202} C_VEL
LIN {X 0,Y 508.597,Z 598.238,A -85,B 0,C 180,E1 18129.831,E2 18129.831} C_VEL
LIN {X 0,Y 508.944,Z 604.723,A -85,B 0,C 180,E1 18129.677,E2 18129.677} C_VEL
LIN {X 0,Y 507.818,Z 613.593,A -85,B 0,C 180,E1 18129.632,E2 18129.632} C_VEL
LIN {X 0,Y 504.867,Z 629.286,A -85,B 0,C 180,E1 18129.65,E2 18129.65} C_VEL
LIN {X 0,Y 504.548,Z 633.806,A -85,B 0,C 180,E1 18129.6,E2 18129.6} C_VEL
LIN {X 0,Y 500.322,Z 851.893,A -85,B 0,C 180,E1 18126.06,E2 18126.06} C_VEL
LIN {X 0,Y 499.316,Z 897.696,A -85,B 0,C 180,E1 18125.285,E2 18125.285} C_VEL
LIN {X 0,Y 498.27,Z 918.107,A -85,B 0,C 180,E1 18124.747,E2 18124.747} C_VEL
LIN {X 0,Y 496.904,Z 938.934,A -85,B 0,C 180,E1 18124.002,E2 18124.002} C_VEL
LIN {X 0,Y 495.317,Z 959.045,A -85,B 0,C 180,E1 18123.07,E2 18123.07} C_VEL
LIN {X 0,Y 493.481,Z 978.788,A -85,B 0,C 180,E1 18121.926,E2 18121.926} C_VEL
LIN {X 0,Y 491.638,Z 997.147,A -85,B 0,C 180,E1 18120.653,E2 18120.653} C_VEL
LIN {X 0,Y 489.353,Z 1019.133,A -85,B 0,C 180,E1 18118.829,E2 18118.829} C_VEL
LIN {X 0,Y 487.575,Z 1036.573,A -85,B 0,C 180,E1 18117.127,E2 18117.127} C_VEL
LIN {X 0,Y 485.837,Z 1053.321,A -85,B 0,C 180,E1 18115.215,E2 18115.215} C_VEL
LIN {X 0,Y 484.358,Z 1068.378,A -85,B 0,C 180,E1 18113.221,E2 18113.221} C_VEL
LIN {X 0,Y 483.023,Z 1082.859,A -85,B 0,C 180,E1 18110.984,E2 18110.984} C_VEL
LIN {X 0,Y 481.979,Z 1095.087,A -85,B 0,C 180,E1 18108.756,E2 18108.756} C_VEL
LIN {X 0,Y 481.13,Z 1106.837,A -85,B 0,C 180,E1 18106.238,E2 18106.238} C_VEL
LIN {X 0,Y 480.589,Z 1116.201,A -85,B 0,C 180,E1 18103.843,E2 18103.843} C_VEL
LIN {X 0,Y 480.236,Z 1123.896,A -85,B 0,C 180,E1 18101.408,E2 18101.408} C_VEL
LIN {X 0,Y 480.032,Z 1130.551,A -85,B 0,C 180,E1 18098.746,E2 18098.746} C_VEL
LIN {X 0,Y 479.942,Z 1135.257,A -85,B 0,C 180,E1 18096.219,E2 18096.219} C_VEL
LIN {X 0,Y 479.905,Z 1138.244,A -85,B 0,C 180,E1 18093.703,E2 18093.703} C_VEL
LIN {X 0,Y 479.907,Z 1139.792,A -85,B 0,C 180,E1 18091.074,E2 18091.074} C_VEL
LIN {X 0,Y 479.908,Z 1139.766,A -85,B 0,C 180,E1 18088.687,E2 18088.687} C_VEL
LIN {X 0,Y 479.908,Z 1138.217,A -85,B 0,C 180,E1 18086.177,E2 18086.177} C_VEL
LIN {X 0,Y 479.945,Z 1135.21,A -85,B 0,C 180,E1 18083.661,E2 18083.661} C_VEL
LIN {X 0,Y 480.032,Z 1130.486,A -85,B 0,C 180,E1 18081.133,E2 18081.133} C_VEL
LIN {X 0,Y 480.236,Z 1123.805,A -85,B 0,C 180,E1 18078.47,E2 18078.47} C_VEL
LIN {X 0,Y 480.593,Z 1116.09,A -85,B 0,C 180,E1 18076.035,E2 18076.035} C_VEL
LIN {X 0,Y 481.152,Z 1106.469,A -85,B 0,C 180,E1 18073.584,E2 18073.584} C_VEL
LIN {X 0,Y 482.009,Z 1094.656,A -85,B 0,C 180,E1 18071.069,E2 18071.069} C_VEL
LIN {X 0,Y 483.106,Z 1081.864,A -85,B 0,C 180,E1 18068.765,E2 18068.765} C_VEL
LIN {X 0,Y 484.385,Z 1068.118,A -85,B 0,C 180,E1 18066.651,E2 18066.651} C_VEL
LIN {X 0,Y 485.918,Z 1052.53,A -85,B 0,C 180,E1 18064.598,E2 18064.598} C_VEL
LIN {X 0,Y 487.684,Z 1035.397,A -85,B 0,C 180,E1 18062.661,E2 18062.661} C_VEL
LIN {X 0,Y 489.517,Z 1017.727,A -85,B 0,C 180,E1 18060.952,E2 18060.952} C_VEL
LIN {X 0,Y 491.85,Z 995.218,A -85,B 0,C 180,E1 18059.109,E2 18059.109} C_VEL
LIN {X 0,Y 493.748,Z 976.175,A -85,B 0,C 180,E1 18057.819,E2 18057.819} C_VEL
LIN {X 0,Y 495.573,Z 955.694,A -85,B 0,C 180,E1 18056.673,E2 18056.673} C_VEL
LIN {X 0,Y 497.237,Z 934.848,A -85,B 0,C 180,E1 18055.743,E2 18055.743} C_VEL
LIN {X 0,Y 498.458,Z 914.783,A -85,B 0,C 180,E1 18055.062,E2 18055.062} C_VEL
LIN {X 0,Y 499.473,Z 892.256,A -85,B 0,C 180,E1 18054.519,E2 18054.519} C_VEL
LIN {X 0,Y 502.833,Z 721.875,A -85,B 0,C 180,E1 18051.733,E2 18051.733} C_VEL
LIN {X 0,Y 504.696,Z 616.817,A -85,B 0,C 180,E1 18050.014,E2 18050.014} C_VEL
LIN {X 0,Y 498.762,Z 587.581,A -85,B 0,C 180,E1 18048.799,E2 18048.799} C_VEL
LIN {X 0,Y 500.288,Z 567.161,A -85,B 0,C 180,E1 18046.881,E2 18046.881} C_VEL
LIN {X 0,Y 493.499,Z 550.748,A -85,B 0,C 180,E1 18044.34,E2 18044.34} C_VEL
LIN {X 0,Y 486.617,Z 535.615,A -85,B 0,C 180,E1 18041.738,E2 18041.738} C_VEL
LIN {X 0,Y 482.074,Z 526.528,A -85,B 0,C 180,E1 18040.013,E2 18040.013} C_VEL
LIN {X 0,Y 480.973,Z 523.822,A -85,B 0,C 180,E1 18039.43,E2 18039.43} C_VEL
LIN {X 0,Y 481.312,Z 524.911,A -85,B 0,C 180,E1 18039.208,E2 18039.208} C_VEL
LIN {X 0,Y 488.533,Z 544.761,A -85,B 0,C 180,E1 18036.993,E2 18036.993} C_VEL
LIN {X 0,Y 491.412,Z 554.051,A -85,B 0,C 180,E1 18036.017,E2 18036.017} C_VEL
LIN {X 0,Y 490.226,Z 597.682,A -85,B 0,C 180,E1 18032.44,E2 18032.44} C_VEL
LIN {X 0,Y 489.02,Z 637.371,A -85,B 0,C 180,E1 18029.184,E2 18029.184} C_VEL
LIN {X 0,Y 487.549,Z 680.634,A -85,B 0,C 180,E1 18025.64,E2 18025.64} C_VEL
LIN {X 0,Y 486.501,Z 711.875,A -85,B 0,C 180,E1 18023.105,E2 18023.105} C_VEL
LIN {X 0,Y 487.559,Z 721.974,A -85,B 0,C 180,E1 18022.886,E2 18022.886} C_VEL
LIN {X 0,Y 485.812,Z 882.293,A -85,B 0,C 180,E1 18020.361,E2 18020.361} C_VEL
LIN {X 0,Y 485.472,Z 899.686,A -85,B 0,C 180,E1 18019.867,E2 18019.867} C_VEL
LIN {X 0,Y 484.962,Z 916.326,A -85,B 0,C 180,E1 18019.171,E2 18019.171} C_VEL
LIN {X 0,Y 484.346,Z 932.457,A -85,B 0,C 180,E1 18018.267,E2 18018.267} C_VEL
LIN {X 0,Y 483.648,Z 947.388,A -85,B 0,C 180,E1 18017.195,E2 18017.195} C_VEL
LIN {X 0,Y 482.935,Z 961.367,A -85,B 0,C 180,E1 18015.932,E2 18015.932} C_VEL
LIN {X 0,Y 482.211,Z 974.563,A -85,B 0,C 180,E1 18014.46,E2 18014.46} C_VEL
LIN {X 0,Y 481.573,Z 986.37,A -85,B 0,C 180,E1 18012.836,E2 18012.836} C_VEL
LIN {X 0,Y 481.066,Z 996.236,A -85,B 0,C 180,E1 18011.145,E2 18011.145} C_VEL
LIN {X 0,Y 480.676,Z 1004.668,A -85,B 0,C 180,E1 18009.338,E2 18009.338} C_VEL
LIN {X 0,Y 480.4,Z 1011.66,A -85,B 0,C 180,E1 18007.414,E2 18007.414} C_VEL
LIN {X 0,Y 480.253,Z 1017.143,A -85,B 0,C 180,E1 18005.376,E2 18005.376} C_VEL
LIN {X 0,Y 480.184,Z 1020.744,A -85,B 0,C 180,E1 18003.343,E2 18003.343} C_VEL
LIN {X 0,Y 480.17,Z 1022.755,A -85,B 0,C 180,E1 18001.193,E2 18001.193} C_VEL
LIN {X 0,Y 480.188,Z 1023.003,A -85,B 0,C 180,E1 17999.046,E2 17999.046} C_VEL
LIN {X 0,Y 480.205,Z 1021.385,A -85,B 0,C 180,E1 17996.897,E2 17996.897} C_VEL
LIN {X 0,Y 480.297,Z 1017.95,A -85,B 0,C 180,E1 17994.745,E2 17994.745} C_VEL
LIN {X 0,Y 480.477,Z 1012.879,A -85,B 0,C 180,E1 17992.708,E2 17992.708} C_VEL
LIN {X 0,Y 480.761,Z 1006.215,A -85,B 0,C 180,E1 17990.785,E2 17990.785} C_VEL
LIN {X 0,Y 481.18,Z 997.522,A -85,B 0,C 180,E1 17988.858,E2 17988.858} C_VEL
LIN {X 0,Y 481.697,Z 987.885,A -85,B 0,C 180,E1 17987.168,E2 17987.168} C_VEL
LIN {X 0,Y 482.311,Z 976.678,A -85,B 0,C 180,E1 17985.596,E2 17985.596} C_VEL
LIN {X 0,Y 482.994,Z 963.885,A -85,B 0,C 180,E1 17984.142,E2 17984.142} C_VEL
LIN {X 0,Y 483.658,Z 949.974,A -85,B 0,C 180,E1 17982.868,E2 17982.868} C_VEL
LIN {X 0,Y 484.264,Z 935.78,A -85,B 0,C 180,E1 17981.835,E2 17981.835} C_VEL
LIN {X 0,Y 484.806,Z 919.613,A -85,B 0,C 180,E1 17980.92,E2 17980.92} C_VEL
LIN {X 0,Y 485.244,Z 902.62,A -85,B 0,C 180,E1 17980.211,E2 17980.211} C_VEL
LIN {X 0,Y 485.49,Z 885.331,A -85,B 0,C 180,E1 17979.727,E2 17979.727} C_VEL
LIN {X 0,Y 487.04,Z 719.12,A -85,B 0,C 180,E1 17977.111,E2 17977.111} C_VEL
LIN {X 0,Y 486.87,Z 716.049,A -85,B 0,C 180,E1 17976.964,E2 17976.964} C_VEL
LIN {X 0,Y 487.867,Z 677.165,A -85,B 0,C 180,E1 17973.922,E2 17973.922} C_VEL
LIN {X 0,Y 488.392,Z 639.865,A -85,B 0,C 180,E1 17971.109,E2 17971.109} C_VEL
LIN {X 0,Y 488.406,Z 603.007,A -85,B 0,C 180,E1 17968.463,E2 17968.463} C_VEL
LIN {X 0,Y 487.898,Z 567.337,A -85,B 0,C 180,E1 17966.06,E2 17966.06} C_VEL
LIN {X 0,Y 487.256,Z 545.161,A -85,B 0,C 180,E1 17964.644,E2 17964.644} C_VEL
LIN {X 0,Y 484.24,Z 533.033,A -85,B 0,C 180,E1 17963.737,E2 17963.737} C_VEL
LIN {X 0,Y 480.948,Z 523.547,A -85,B 0,C 180,E1 17962.923,E2 17962.923} C_VEL
LIN {X 0,Y 480.861,Z 523.178,A -85,B 0,C 180,E1 17962.394,E2 17962.394} C_VEL
LIN {X 0,Y 480.929,Z 523.614,A -85,B 0,C 180,E1 17962.089,E2 17962.089} C_VEL
LIN {X 0,Y 482.564,Z 527.109,A -85,B 0,C 180,E1 17961.416,E2 17961.416} C_VEL
LIN {X 0,Y 487.846,Z 537.913,A -85,B 0,C 180,E1 17959.481,E2 17959.481} C_VEL
LIN {X 0,Y 492.711,Z 547.911,A -85,B 0,C 180,E1 17957.842,E2 17957.842} C_VEL
LIN {X 0,Y 506.538,Z 568.636,A -85,B 0,C 180,E1 17955.87,E2 17955.87} C_VEL
LIN {X 0,Y 509.622,Z 573.772,A -85,B 0,C 180,E1 17955.448,E2 17955.448} C_VEL
LIN {X 0,Y 505.514,Z 779.507,A -85,B 0,C 180,E1 17952.004,E2 17952.004} C_VEL
LIN {X 0,Y 503.433,Z 893.119,A -85,B 0,C 180,E1 17950.144,E2 17950.144} C_VEL
LIN {X 0,Y 502.404,Z 915.774,A -85,B 0,C 180,E1 17949.587,E2 17949.587} C_VEL
LIN {X 0,Y 501.161,Z 937.535,A -85,B 0,C 180,E1 17948.872,E2 17948.872} C_VEL
LIN {X 0,Y 499.486,Z 959.866,A -85,B 0,C 180,E1 17947.919,E2 17947.919} C_VEL
LIN {X 0,Y 497.713,Z 981.698,A -85,B 0,C 180,E1 17946.774,E2 17946.774} C_VEL
LIN {X 0,Y 495.819,Z 1000.12,A -85,B 0,C 180,E1 17945.576,E2 17945.576} C_VEL
LIN {X 0,Y 493.622,Z 1020.167,A -85,B 0,C 180,E1 17944.061,E2 17944.061} C_VEL
LIN {X 0,Y 491.392,Z 1039.257,A -85,B 0,C 180,E1 17942.354,E2 17942.354} C_VEL
LIN {X 0,Y 489.089,Z 1058.781,A -85,B 0,C 180,E1 17940.328,E2 17940.328} C_VEL
LIN {X 0,Y 487.196,Z 1075.148,A -85,B 0,C 180,E1 17938.366,E2 17938.366} C_VEL
LIN {X 0,Y 485.379,Z 1091.137,A -85,B 0,C 180,E1 17936.157,E2 17936.157} C_VEL
LIN {X 0,Y 483.812,Z 1106.227,A -85,B 0,C 180,E1 17933.765,E2 17933.765} C_VEL
LIN {X 0,Y 482.571,Z 1119.082,A -85,B 0,C 180,E1 17931.387,E2 17931.387} C_VEL
LIN {X 0,Y 481.559,Z 1131.29,A -85,B 0,C 180,E1 17928.773,E2 17928.773} C_VEL
LIN {X 0,Y 480.878,Z 1141.065,A -85,B 0,C 180,E1 17926.302,E2 17926.302} C_VEL
LIN {X 0,Y 480.379,Z 1150.348,A -85,B 0,C 180,E1 17923.481,E2 17923.481} C_VEL
LIN {X 0,Y 480.127,Z 1157.168,A -85,B 0,C 180,E1 17920.924,E2 17920.924} C_VEL
LIN {X 0,Y 479.98,Z 1162.635,A -85,B 0,C 180,E1 17918.264,E2 17918.264} C_VEL
LIN {X 0,Y 479.907,Z 1166.437,A -85,B 0,C 180,E1 17915.74,E2 17915.74} C_VEL
LIN {X 0,Y 479.889,Z 1168.986,A -85,B 0,C 180,E1 17912.986,E2 17912.986} C_VEL
LIN {X 0,Y 479.884,Z 1169.895,A -85,B 0,C 180,E1 17910.597,E2 17910.597} C_VEL
LIN {X 0,Y 479.913,Z 1169.393,A -85,B 0,C 180,E1 17907.731,E2 17907.731} C_VEL
LIN {X 0,Y 479.911,Z 1167.501,A -85,B 0,C 180,E1 17905.22,E2 17905.22} C_VEL
LIN {X 0,Y 479.943,Z 1163.874,A -85,B 0,C 180,E1 17902.458,E2 17902.458} C_VEL
LIN {X 0,Y 480.027,Z 1159.508,A -85,B 0,C 180,E1 17900.134,E2 17900.134} C_VEL
LIN {X 0,Y 480.254,Z 1153.172,A -85,B 0,C 180,E1 17897.495,E2 17897.495} C_VEL
LIN {X 0,Y 480.636,Z 1145.341,A -85,B 0,C 180,E1 17894.928,E2 17894.928} C_VEL
LIN {X 0,Y 481.268,Z 1135.417,A -85,B 0,C 180,E1 17892.218,E2 17892.218} C_VEL
LIN {X 0,Y 482.1,Z 1124.576,A -85,B 0,C 180,E1 17889.736,E2 17889.736} C_VEL
LIN {X 0,Y 483.311,Z 1111.15,A -85,B 0,C 180,E1 17887.112,E2 17887.112} C_VEL
LIN {X 0,Y 484.766,Z 1097.015,A -85,B 0,C 180,E1 17884.726,E2 17884.726} C_VEL
LIN {X 0,Y 486.457,Z 1081.331,A -85,B 0,C 180,E1 17882.454,E2 17882.454} C_VEL
LIN {X 0,Y 488.453,Z 1064.331,A -85,B 0,C 180,E1 17880.306,E2 17880.306} C_VEL
LIN {X 0,Y 490.425,Z 1047.391,A -85,B 0,C 180,E1 17878.451,E2 17878.451} C_VEL
LIN {X 0,Y 492.764,Z 1027.511,A -85,B 0,C 180,E1 17876.571,E2 17876.571} C_VEL
LIN {X 0,Y 494.865,Z 1008.884,A -85,B 0,C 180,E1 17875.054,E2 17875.054} C_VEL
LIN {X 0,Y 496.993,Z 988.816,A -85,B 0,C 180,E1 17873.667,E2 17873.667} C_VEL
LIN {X 0,Y 498.488,Z 972.464,A -85,B 0,C 180,E1 17872.717,E2 17872.717} C_VEL
LIN {X 0,Y 500.271,Z 950.189,A -85,B 0,C 180,E1 17871.642,E2 17871.642} C_VEL
LIN {X 0,Y 501.653,Z 928.879,A -85,B 0,C 180,E1 17870.822,E2 17870.822} C_VEL
LIN {X 0,Y 502.937,Z 904.439,A -85,B 0,C 180,E1 17870.11,E2 17870.11} C_VEL
LIN {X 0,Y 503.754,Z 882.018,A -85,B 0,C 180,E1 17869.655,E2 17869.655} C_VEL
LIN {X 0,Y 507.465,Z 675.958,A -85,B 0,C 180,E1 17866.284,E2 17866.284} C_VEL
LIN {X 0,Y 509.561,Z 571.689,A -85,B 0,C 180,E1 17864.51,E2 17864.51} C_VEL
LIN {X 0,Y 494.257,Z 548.785,A -85,B 0,C 180,E1 17862.368,E2 17862.368} C_VEL
LIN {X 0,Y 492.27,Z 545.46,A -85,B 0,C 180,E1 17862.001,E2 17862.001} C_VEL
LIN {X 0,Y 485.134,Z 531.823,A -85,B 0,C 180,E1 17859.864,E2 17859.864} C_VEL
LIN {X 0,Y 482.903,Z 527.524,A -85,B 0,C 180,E1 17859.161,E2 17859.161} C_VEL
LIN {X 0,Y 481.075,Z 524.181,A -85,B 0,C 180,E1 17858.573,E2 17858.573} C_VEL
LIN {X 0,Y 480.894,Z 523.24,A -85,B 0,C 180,E1 17858.337,E2 17858.337} C_VEL
LIN {X 0,Y 480.884,Z 523.148,A -85,B 0,C 180,E1 17854.729,E2 17854.729} C_VEL
LIN {X 0,Y 480.879,Z 523.126,A -85,B 0,C 180,E1 17851.18,E2 17851.18} C_VEL
LIN {X 0,Y 480.884,Z 523.113,A -85,B 0,C 180,E1 17847.623,E2 17847.623} C_VEL
LIN {X 0,Y 480.879,Z 523.148,A -85,B 0,C 180,E1 17843.919,E2 17843.919} C_VEL
LIN {X 0,Y 480.882,Z 523.124,A -85,B 0,C 180,E1 17840.326,E2 17840.326} C_VEL
LIN {X 0,Y 480.879,Z 523.121,A -85,B 0,C 180,E1 17836.674,E2 17836.674} C_VEL
LIN {X 0,Y 480.879,Z 523.135,A -85,B 0,C 180,E1 17833.099,E2 17833.099} C_VEL
LIN {X 0,Y 480.884,Z 523.11,A -85,B 0,C 180,E1 17829.454,E2 17829.454} C_VEL
LIN {X 0,Y 480.876,Z 523.147,A -85,B 0,C 180,E1 17825.847,E2 17825.847} C_VEL
LIN {X 0,Y 480.886,Z 523.142,A -85,B 0,C 180,E1 17822.264,E2 17822.264} C_VEL
LIN {X 0,Y 480.885,Z 523.141,A -85,B 0,C 180,E1 17818.689,E2 17818.689} C_VEL
LIN {X 0,Y 480.876,Z 523.146,A -85,B 0,C 180,E1 17815.109,E2 17815.109} C_VEL
LIN {X 0,Y 480.886,Z 523.144,A -85,B 0,C 180,E1 17811.51,E2 17811.51} C_VEL
LIN {X 0,Y 480.879,Z 523.109,A -85,B 0,C 180,E1 17807.877,E2 17807.877} C_VEL
LIN {X 0,Y 480.883,Z 523.145,A -85,B 0,C 180,E1 17804.298,E2 17804.298} C_VEL
LIN {X 0,Y 480.87,Z 523.109,A -85,B 0,C 180,E1 17800.694,E2 17800.694} C_VEL
LIN {X 0,Y 480.887,Z 523.146,A -85,B 0,C 180,E1 17797.086,E2 17797.086} C_VEL
LIN {X 0,Y 480.888,Z 523.123,A -85,B 0,C 180,E1 17793.388,E2 17793.388} C_VEL
LIN {X 0,Y 480.867,Z 523.119,A -85,B 0,C 180,E1 17789.881,E2 17789.881} C_VEL
LIN {X 0,Y 480.886,Z 523.146,A -85,B 0,C 180,E1 17786.272,E2 17786.272} C_VEL
LIN {X 0,Y 480.886,Z 523.135,A -85,B 0,C 180,E1 17782.585,E2 17782.585} C_VEL
LIN {X 0,Y 480.901,Z 523.368,A -85,B 0,C 180,E1 17779.192,E2 17779.192} C_VEL
LIN {X 0,Y 482.266,Z 526.714,A -85,B 0,C 180,E1 17778.596,E2 17778.596} C_VEL
LIN {X 0,Y 483.427,Z 528.645,A -85,B 0,C 180,E1 17778.242,E2 17778.242} C_VEL
LIN {X 0,Y 490.194,Z 542.044,A -85,B 0,C 180,E1 17776.056,E2 17776.056} C_VEL
LIN {X 0,Y 498.2,Z 558.804,A -85,B 0,C 180,E1 17773.572,E2 17773.572} C_VEL
LIN {X 0,Y 501.963,Z 567.496,A -85,B 0,C 180,E1 17772.397,E2 17772.397} C_VEL
LIN {X 0,Y 500.579,Z 587.744,A -85,B 0,C 180,E1 17770.876,E2 17770.876} C_VEL
LIN {X 0,Y 504.921,Z 614.59,A -85,B 0,C 180,E1 17769.913,E2 17769.913} C_VEL
LIN {X 0,Y 504.548,Z 633.806,A -85,B 0,C 180,E1 17769.6,E2 17769.6} C_VEL
LIN {X 0,Y 503.67,Z 641.509,A -85,B 0,C 180,E1 17769.551,E2 17769.551} C_VEL
LIN {X 0,Y 498.63,Z 662.112,A -85,B 0,C 180,E1 17769.699,E2 17769.699} C_VEL
LIN {X 0,Y 497.934,Z 668.724,A -85,B 0,C 180,E1 17769.651,E2 17769.651} C_VEL
LIN {X 0,Y 493.728,Z 879.176,A -85,B 0,C 180,E1 17766.221,E2 17766.221} C_VEL
LIN {X 0,Y 492.89,Z 903.436,A -85,B 0,C 180,E1 17765.749,E2 17765.749} C_VEL
LIN {X 0,Y 491.727,Z 924.083,A -85,B 0,C 180,E1 17765.16,E2 17765.16} C_VEL
LIN {X 0,Y 490.207,Z 944.357,A -85,B 0,C 180,E1 17764.363,E2 17764.363} C_VEL
LIN {X 0,Y 488.385,Z 964.602,A -85,B 0,C 180,E1 17763.354,E2 17763.354} C_VEL
LIN {X 0,Y 486.406,Z 984.015,A -85,B 0,C 180,E1 17762.168,E2 17762.168} C_VEL
LIN {X 0,Y 484.335,Z 1002.484,A -85,B 0,C 180,E1 17760.795,E2 17760.795} C_VEL
LIN {X 0,Y 482.045,Z 1021.718,A -85,B 0,C 180,E1 17759.104,E2 17759.104} C_VEL
LIN {X 0,Y 479.901,Z 1039.921,A -85,B 0,C 180,E1 17757.214,E2 17757.214} C_VEL
LIN {X 0,Y 478.072,Z 1056.366,A -85,B 0,C 180,E1 17755.255,E2 17755.255} C_VEL
LIN {X 0,Y 476.48,Z 1071.125,A -85,B 0,C 180,E1 17753.203,E2 17753.203} C_VEL
LIN {X 0,Y 475.111,Z 1085.009,A -85,B 0,C 180,E1 17750.963,E2 17750.963} C_VEL
LIN {X 0,Y 473.991,Z 1097.632,A -85,B 0,C 180,E1 17748.574,E2 17748.574} C_VEL
LIN {X 0,Y 473.169,Z 1108.157,A -85,B 0,C 180,E1 17746.196,E2 17746.196} C_VEL
LIN {X 0,Y 472.571,Z 1117.831,A -85,B 0,C 180,E1 17743.583,E2 17743.583} C_VEL
LIN {X 0,Y 472.223,Z 1125.311,A -85,B 0,C 180,E1 17741.109,E2 17741.109} C_VEL
LIN {X 0,Y 472.024,Z 1131.316,A -85,B 0,C 180,E1 17738.527,E2 17738.527} C_VEL
LIN {X 0,Y 471.934,Z 1135.902,A -85,B 0,C 180,E1 17735.837,E2 17735.837} C_VEL
LIN {X 0,Y 471.907,Z 1138.696,A -85,B 0,C 180,E1 17733.279,E2 17733.279} C_VEL
LIN {X 0,Y 471.899,Z 1139.86,A -85,B 0,C 180,E1 17730.728,E2 17730.728} C_VEL
LIN {X 0,Y 471.901,Z 1139.609,A -85,B 0,C 180,E1 17728.179,E2 17728.179} C_VEL
LIN {X 0,Y 471.921,Z 1137.761,A -85,B 0,C 180,E1 17725.626,E2 17725.626} C_VEL
LIN {X 0,Y 471.954,Z 1134.181,A -85,B 0,C 180,E1 17722.942,E2 17722.942} C_VEL
LIN {X 0,Y 472.067,Z 1129.467,A -85,B 0,C 180,E1 17720.491,E2 17720.491} C_VEL
LIN {X 0,Y 472.302,Z 1122.945,A -85,B 0,C 180,E1 17717.974,E2 17717.974} C_VEL
LIN {X 0,Y 472.734,Z 1114.72,A -85,B 0,C 180,E1 17715.422,E2 17715.422} C_VEL
LIN {X 0,Y 473.402,Z 1104.913,A -85,B 0,C 180,E1 17712.928,E2 17712.928} C_VEL
LIN {X 0,Y 474.313,Z 1093.633,A -85,B 0,C 180,E1 17710.545,E2 17710.545} C_VEL
LIN {X 0,Y 475.555,Z 1080.315,A -85,B 0,C 180,E1 17708.152,E2 17708.152} C_VEL
LIN {X 0,Y 477.012,Z 1066.393,A -85,B 0,C 180,E1 17706.006,E2 17706.006} C_VEL
LIN {X 0,Y 478.66,Z 1050.969,A -85,B 0,C 180,E1 17703.981,E2 17703.981} C_VEL
LIN {X 0,Y 480.894,Z 1031.329,A -85,B 0,C 180,E1 17701.77,E2 17701.77} C_VEL
LIN {X 0,Y 483.083,Z 1013.085,A -85,B 0,C 180,E1 17700.01,E2 17700.01} C_VEL
LIN {X 0,Y 485.221,Z 994.849,A -85,B 0,C 180,E1 17698.515,E2 17698.515} C_VEL
LIN {X 0,Y 487.179,Z 976.625,A -85,B 0,C 180,E1 17697.269,E2 17697.269} C_VEL
LIN {X 0,Y 489.218,Z 955.562,A -85,B 0,C 180,E1 17696.076,E2 17696.076} C_VEL
LIN {X 0,Y 490.984,Z 934.969,A -85,B 0,C 180,E1 17695.151,E2 17695.151} C_VEL
LIN {X 0,Y 492.286,Z 914.875,A -85,B 0,C 180,E1 17694.465,E2 17694.465} C_VEL
LIN {X 0,Y 493.365,Z 892.16,A -85,B 0,C 180,E1 17693.917,E2 17693.917} C_VEL
LIN {X 0,Y 496.942,Z 717.53,A -85,B 0,C 180,E1 17691.048,E2 17691.048} C_VEL
LIN {X 0,Y 498.796,Z 618.574,A -85,B 0,C 180,E1 17689.418,E2 17689.418} C_VEL
LIN {X 0,Y 492.449,Z 587.161,A -85,B 0,C 180,E1 17688.087,E2 17688.087} C_VEL
LIN {X 0,Y 493.72,Z 571.038,A -85,B 0,C 180,E1 17686.554,E2 17686.554} C_VEL
LIN {X 0,Y 487.261,Z 555.32,A -85,B 0,C 180,E1 17684.078,E2 17684.078} C_VEL
LIN {X 0,Y 480.58,Z 540.569,A -85,B 0,C 180,E1 17681.497,E2 17681.497} C_VEL
LIN {X 0,Y 476.181,Z 531.646,A -85,B 0,C 180,E1 17679.78,E2 17679.78} C_VEL
LIN {X 0,Y 475.412,Z 529.997,A -85,B 0,C 180,E1 17679.431,E2 17679.431} C_VEL
LIN {X 0,Y 475.27,Z 530.452,A -85,B 0,C 180,E1 17679.221,E2 17679.221} C_VEL
LIN {X 0,Y 483.373,Z 553.575,A -85,B 0,C 180,E1 17676.622,E2 17676.622} C_VEL
LIN {X 0,Y 484.191,Z 557.032,A -85,B 0,C 180,E1 17676.273,E2 17676.273} C_VEL
LIN {X 0,Y 482.914,Z 601.131,A -85,B 0,C 180,E1 17672.64,E2 17672.64} C_VEL
LIN {X 0,Y 481.613,Z 641.426,A -85,B 0,C 180,E1 17669.314,E2 17669.314} C_VEL
LIN {X 0,Y 480.066,Z 684.823,A -85,B 0,C 180,E1 17665.738,E2 17665.738} C_VEL
LIN {X 0,Y 479.09,Z 712.917,A -85,B 0,C 180,E1 17663.446,E2 17663.446} C_VEL
LIN {X 0,Y 480.124,Z 722.974,A -85,B 0,C 180,E1 17663.225,E2 17663.225} C_VEL
LIN {X 0,Y 478.209,Z 883.564,A -85,B 0,C 180,E1 17660.636,E2 17660.636} C_VEL
LIN {X 0,Y 477.861,Z 900.938,A -85,B 0,C 180,E1 17660.133,E2 17660.133} C_VEL
LIN {X 0,Y 477.354,Z 917.018,A -85,B 0,C 180,E1 17659.454,E2 17659.454} C_VEL
LIN {X 0,Y 476.711,Z 933.298,A -85,B 0,C 180,E1 17658.534,E2 17658.534} C_VEL
LIN {X 0,Y 475.969,Z 948.671,A -85,B 0,C 180,E1 17657.419,E2 17657.419} C_VEL
LIN {X 0,Y 475.218,Z 962.77,A -85,B 0,C 180,E1 17656.125,E2 17656.125} C_VEL
LIN {X 0,Y 474.444,Z 976.321,A -85,B 0,C 180,E1 17654.587,E2 17654.587} C_VEL
LIN {X 0,Y 473.771,Z 988.122,A -85,B 0,C 180,E1 17652.927,E2 17652.927} C_VEL
LIN {X 0,Y 473.235,Z 997.92,A -85,B 0,C 180,E1 17651.209,E2 17651.209} C_VEL
LIN {X 0,Y 472.806,Z 1006.822,A -85,B 0,C 180,E1 17649.249,E2 17649.249} C_VEL
LIN {X 0,Y 472.532,Z 1013.678,A -85,B 0,C 180,E1 17647.294,E2 17647.294} C_VEL
LIN {X 0,Y 472.367,Z 1018.935,A -85,B 0,C 180,E1 17645.222,E2 17645.222} C_VEL
LIN {X 0,Y 472.3,Z 1022.572,A -85,B 0,C 180,E1 17643.034,E2 17643.034} C_VEL
LIN {X 0,Y 472.3,Z 1024.305,A -85,B 0,C 180,E1 17640.971,E2 17640.971} C_VEL
LIN {X 0,Y 472.319,Z 1024.383,A -85,B 0,C 180,E1 17638.909,E2 17638.909} C_VEL
LIN {X 0,Y 472.352,Z 1022.689,A -85,B 0,C 180,E1 17636.724,E2 17636.724} C_VEL
LIN {X 0,Y 472.457,Z 1019.4,A -85,B 0,C 180,E1 17634.657,E2 17634.657} C_VEL
LIN {X 0,Y 472.648,Z 1014.66,A -85,B 0,C 180,E1 17632.708,E2 17632.708} C_VEL
LIN {X 0,Y 472.95,Z 1008.074,A -85,B 0,C 180,E1 17630.755,E2 17630.755} C_VEL
LIN {X 0,Y 473.393,Z 999.44,A -85,B 0,C 180,E1 17628.796,E2 17628.796} C_VEL
LIN {X 0,Y 473.935,Z 989.862,A -85,B 0,C 180,E1 17627.078,E2 17627.078} C_VEL
LIN {X 0,Y 474.574,Z 978.733,A -85,B 0,C 180,E1 17625.481,E2 17625.481} C_VEL
LIN {X 0,Y 475.28,Z 965.98,A -85,B 0,C 180,E1 17624.003,E2 17624.003} C_VEL
LIN {X 0,Y 475.969,Z 952.075,A -85,B 0,C 180,E1 17622.703,E2 17622.703} C_VEL
LIN {X 0,Y 476.58,Z 938.06,A -85,B 0,C 180,E1 17621.658,E2 17621.658} C_VEL
LIN {X 0,Y 477.12,Z 922.335,A -85,B 0,C 180,E1 17620.745,E2 17620.745} C_VEL
LIN {X 0,Y 477.566,Z 905.063,A -85,B 0,C 180,E1 17620.003,E2 17620.003} C_VEL
LIN {X 0,Y 477.809,Z 887.866,A -85,B 0,C 180,E1 17619.502,E2 17619.502} C_VEL
LIN {X 0,Y 479.61,Z 724.846,A -85,B 0,C 180,E1 17616.869,E2 17616.869} C_VEL
LIN {X 0,Y 479.563,Z 719.69,A -85,B 0,C 180,E1 17616.761,E2 17616.761} C_VEL
LIN {X 0,Y 480.617,Z 675.971,A -85,B 0,C 180,E1 17613.365,E2 17613.365} C_VEL
LIN {X 0,Y 481.132,Z 637.708,A -85,B 0,C 180,E1 17610.494,E2 17610.494} C_VEL
LIN {X 0,Y 481.09,Z 601.875,A -85,B 0,C 180,E1 17607.934,E2 17607.934} C_VEL
LIN {X 0,Y 480.578,Z 564.004,A -85,B 0,C 180,E1 17605.391,E2 17605.391} C_VEL
LIN {X 0,Y 479.988,Z 547.351,A -85,B 0,C 180,E1 17604.32,E2 17604.32} C_VEL
LIN {X 0,Y 477.262,Z 536.262,A -85,B 0,C 180,E1 17603.469,E2 17603.469} C_VEL
LIN {X 0,Y 474.425,Z 527.924,A -85,B 0,C 180,E1 17602.725,E2 17602.725} C_VEL
LIN {X 0,Y 474.419,Z 527.89,A -85,B 0,C 180,E1 17602.554,E2 17602.554} C_VEL
LIN {X 0,Y 475.517,Z 529.959,A -85,B 0,C 180,E1 17602.123,E2 17602.123} C_VEL
LIN {X 0,Y 479.766,Z 538.383,A -85,B 0,C 180,E1 17600.533,E2 17600.533} C_VEL
LIN {X 0,Y 484.699,Z 548.584,A -85,B 0,C 180,E1 17598.791,E2 17598.791} C_VEL
LIN {X 0,Y 496.012,Z 565.216,A -85,B 0,C 180,E1 17597.092,E2 17597.092} C_VEL
LIN {X 0,Y 503.652,Z 577.221,A -85,B 0,C 180,E1 17596.007,E2 17596.007} C_VEL
LIN {X 0,Y 499.086,Z 787.404,A -85,B 0,C 180,E1 17592.443,E2 17592.443} C_VEL
LIN {X 0,Y 496.932,Z 893.447,A -85,B 0,C 180,E1 17590.677,E2 17590.677} C_VEL
LIN {X 0,Y 495.829,Z 915.977,A -85,B 0,C 180,E1 17590.115,E2 17590.115} C_VEL
LIN {X 0,Y 494.482,Z 938.093,A -85,B 0,C 180,E1 17589.377,E2 17589.377} C_VEL
LIN {X 0,Y 492.755,Z 959.661,A -85,B 0,C 180,E1 17588.443,E2 17588.443} C_VEL
LIN {X 0,Y 490.874,Z 981.295,A -85,B 0,C 180,E1 17587.299,E2 17587.299} C_VEL
LIN {X 0,Y 488.87,Z 1001.347,A -85,B 0,C 180,E1 17586.016,E2 17586.016} C_VEL
LIN {X 0,Y 486.917,Z 1019.421,A -85,B 0,C 180,E1 17584.667,E2 17584.667} C_VEL
LIN {X 0,Y 484.479,Z 1038.587,A -85,B 0,C 180,E1 17582.943,E2 17582.943} C_VEL
LIN {X 0,Y 482.084,Z 1057.67,A -85,B 0,C 180,E1 17580.955,E2 17580.955} C_VEL
LIN {X 0,Y 479.98,Z 1074.151,A -85,B 0,C 180,E1 17578.966,E2 17578.966} C_VEL
LIN {X 0,Y 478.016,Z 1090.29,A -85,B 0,C 180,E1 17576.725,E2 17576.725} C_VEL
LIN {X 0,Y 476.313,Z 1105.172,A -85,B 0,C 180,E1 17574.352,E2 17574.352} C_VEL
LIN {X 0,Y 474.893,Z 1118.445,A -85,B 0,C 180,E1 17571.88,E2 17571.88} C_VEL
LIN {X 0,Y 473.821,Z 1130.249,A -85,B 0,C 180,E1 17569.348,E2 17569.348} C_VEL
LIN {X 0,Y 473.027,Z 1140.409,A -85,B 0,C 180,E1 17566.761,E2 17566.761} C_VEL
LIN {X 0,Y 472.461,Z 1149.638,A -85,B 0,C 180,E1 17563.961,E2 17563.961} C_VEL
LIN {X 0,Y 472.171,Z 1156.259,A -85,B 0,C 180,E1 17561.482,E2 17561.482} C_VEL
LIN {X 0,Y 472.003,Z 1162.222,A -85,B 0,C 180,E1 17558.65,E2 17558.65} C_VEL
LIN {X 0,Y 471.918,Z 1166.119,A -85,B 0,C 180,E1 17556.081,E2 17556.081} C_VEL
LIN {X 0,Y 471.886,Z 1168.849,A -85,B 0,C 180,E1 17553.28,E2 17553.28} C_VEL
LIN {X 0,Y 471.887,Z 1169.849,A -85,B 0,C 180,E1 17550.85,E2 17550.85} C_VEL
LIN {X 0,Y 471.905,Z 1169.658,A -85,B 0,C 180,E1 17548.179,E2 17548.179} C_VEL
LIN {X 0,Y 471.91,Z 1167.842,A -85,B 0,C 180,E1 17545.504,E2 17545.504} C_VEL
LIN {X 0,Y 471.927,Z 1164.681,A -85,B 0,C 180,E1 17542.819,E2 17542.819} C_VEL
LIN {X 0,Y 472.03,Z 1160.082,A -85,B 0,C 180,E1 17540.244,E2 17540.244} C_VEL
LIN {X 0,Y 472.244,Z 1154.437,A -85,B 0,C 180,E1 17537.776,E2 17537.776} C_VEL
LIN {X 0,Y 472.667,Z 1146.15,A -85,B 0,C 180,E1 17534.919,E2 17534.919} C_VEL
LIN {X 0,Y 473.301,Z 1136.922,A -85,B 0,C 180,E1 17532.29,E2 17532.29} C_VEL
LIN {X 0,Y 474.219,Z 1125.721,A -85,B 0,C 180,E1 17529.642,E2 17529.642} C_VEL
LIN {X 0,Y 475.456,Z 1113.142,A -85,B 0,C 180,E1 17527.085,E2 17527.085} C_VEL
LIN {X 0,Y 476.953,Z 1099.341,A -85,B 0,C 180,E1 17524.681,E2 17524.681} C_VEL
LIN {X 0,Y 478.852,Z 1083.181,A -85,B 0,C 180,E1 17522.249,E2 17522.249} C_VEL
LIN {X 0,Y 480.98,Z 1066.529,A -85,B 0,C 180,E1 17520.072,E2 17520.072} C_VEL
LIN {X 0,Y 483.197,Z 1048.713,A -85,B 0,C 180,E1 17518.076,E2 17518.076} C_VEL
LIN {X 0,Y 485.627,Z 1029.711,A -85,B 0,C 180,E1 17516.227,E2 17516.227} C_VEL
LIN {X 0,Y 487.635,Z 1012.857,A -85,B 0,C 180,E1 17514.818,E2 17514.818} C_VEL
LIN {X 0,Y 489.751,Z 992.829,A -85,B 0,C 180,E1 17513.406,E2 17513.406} C_VEL
LIN {X 0,Y 491.715,Z 972.024,A -85,B 0,C 180,E1 17512.188,E2 17512.188} C_VEL
LIN {X 0,Y 493.596,Z 949.676,A -85,B 0,C 180,E1 17511.1,E2 17511.1} C_VEL
LIN {X 0,Y 495.077,Z 928.224,A -85,B 0,C 180,E1 17510.27,E2 17510.27} C_VEL
LIN {X 0,Y 496.431,Z 904.202,A -85,B 0,C 180,E1 17509.568,E2 17509.568} C_VEL
LIN {X 0,Y 497.298,Z 881.611,A -85,B 0,C 180,E1 17509.105,E2 17509.105} C_VEL
LIN {X 0,Y 501.054,Z 690.708,A -85,B 0,C 180,E1 17505.938,E2 17505.938} C_VEL
LIN {X 0,Y 503.565,Z 575.216,A -85,B 0,C 180,E1 17503.943,E2 17503.943} C_VEL
LIN {X 0,Y 489.3,Z 553.734,A -85,B 0,C 180,E1 17501.889,E2 17501.889} C_VEL
LIN {X 0,Y 484.643,Z 546.767,A -85,B 0,C 180,E1 17501.147,E2 17501.147} C_VEL
LIN {X 0,Y 477.445,Z 533.134,A -85,B 0,C 180,E1 17498.921,E2 17498.921} C_VEL
LIN {X 0,Y 474.853,Z 528.407,A -85,B 0,C 180,E1 17498.093,E2 17498.093} C_VEL
LIN {X 0,Y 473.079,Z 524.894,A -85,B 0,C 180,E1 17497.461,E2 17497.461} C_VEL
LIN {X 0,Y 472.96,Z 524.216,A -85,B 0,C 180,E1 17497.201,E2 17497.201} C_VEL
LIN {X 0,Y 472.942,Z 524.111,A -85,B 0,C 180,E1 17493.489,E2 17493.489} C_VEL
LIN {X 0,Y 472.948,Z 524.139,A -85,B 0,C 180,E1 17489.789,E2 17489.789} C_VEL
LIN {X 0,Y 472.938,Z 524.112,A -85,B 0,C 180,E1 17486.087,E2 17486.087} C_VEL
LIN {X 0,Y 472.94,Z 524.103,A -85,B 0,C 180,E1 17482.498,E2 17482.498} C_VEL
LIN {X 0,Y 472.946,Z 524.136,A -85,B 0,C 180,E1 17478.872,E2 17478.872} C_VEL
LIN {X 0,Y 472.937,Z 524.092,A -85,B 0,C 180,E1 17475.198,E2 17475.198} C_VEL
LIN {X 0,Y 472.948,Z 524.131,A -85,B 0,C 180,E1 17471.586,E2 17471.586} C_VEL
LIN {X 0,Y 472.934,Z 524.096,A -85,B 0,C 180,E1 17467.898,E2 17467.898} C_VEL
LIN {X 0,Y 472.945,Z 524.13,A -85,B 0,C 180,E1 17464.243,E2 17464.243} C_VEL
LIN {X 0,Y 472.944,Z 524.133,A -85,B 0,C 180,E1 17460.605,E2 17460.605} C_VEL
LIN {X 0,Y 472.944,Z 524.129,A -85,B 0,C 180,E1 17456.97,E2 17456.97} C_VEL
LIN {X 0,Y 472.936,Z 524.127,A -85,B 0,C 180,E1 17453.322,E2 17453.322} C_VEL
LIN {X 0,Y 472.945,Z 524.127,A -85,B 0,C 180,E1 17449.771,E2 17449.771} C_VEL
LIN {X 0,Y 472.947,Z 524.108,A -85,B 0,C 180,E1 17446.02,E2 17446.02} C_VEL
LIN {X 0,Y 472.934,Z 524.12,A -85,B 0,C 180,E1 17442.402,E2 17442.402} C_VEL
LIN {X 0,Y 472.938,Z 524.125,A -85,B 0,C 180,E1 17438.676,E2 17438.676} C_VEL
LIN {X 0,Y 472.943,Z 524.099,A -85,B 0,C 180,E1 17435.089,E2 17435.089} C_VEL
LIN {X 0,Y 472.954,Z 524.134,A -85,B 0,C 180,E1 17431.459,E2 17431.459} C_VEL
LIN {X 0,Y 472.929,Z 524.114,A -85,B 0,C 180,E1 17427.807,E2 17427.807} C_VEL
LIN {X 0,Y 472.943,Z 524.101,A -85,B 0,C 180,E1 17424.153,E2 17424.153} C_VEL
LIN {X 0,Y 472.953,Z 524.169,A -85,B 0,C 180,E1 17420.48,E2 17420.48} C_VEL
LIN {X 0,Y 473.041,Z 524.679,A -85,B 0,C 180,E1 17420.175,E2 17420.175} C_VEL
LIN {X 0,Y 474.642,Z 528.146,A -85,B 0,C 180,E1 17419.547,E2 17419.547} C_VEL
LIN {X 0,Y 478.46,Z 535.515,A -85,B 0,C 180,E1 17418.249,E2 17418.249} C_VEL
LIN {X 0,Y 484.201,Z 546.594,A -85,B 0,C 180,E1 17416.393,E2 17416.393} C_VEL
LIN {X 0,Y 492.973,Z 565.276,A -85,B 0,C 180,E1 17413.598,E2 17413.598} C_VEL
LIN {X 0,Y 495.53,Z 571.208,A -85,B 0,C 180,E1 17412.785,E2 17412.785} C_VEL
LIN {X 0,Y 494.371,Z 587.116,A -85,B 0,C 180,E1 17411.577,E2 17411.577} C_VEL
LIN {X 0,Y 499.021,Z 616.064,A -85,B 0,C 180,E1 17410.514,E2 17410.514} C_VEL
LIN {X 0,Y 497.934,Z 668.724,A -85,B 0,C 180,E1 17409.651,E2 17409.651} C_VEL
LIN {X 0,Y 497.042,Z 676.428,A -85,B 0,C 180,E1 17409.604,E2 17409.604} C_VEL
LIN {X 0,Y 492.026,Z 697.032,A -85,B 0,C 180,E1 17409.76,E2 17409.76} C_VEL
LIN {X 0,Y 491.329,Z 703.643,A -85,B 0,C 180,E1 17409.712,E2 17409.712} C_VEL
LIN {X 0,Y 487.307,Z 892.153,A -85,B 0,C 180,E1 17406.608,E2 17406.608} C_VEL
LIN {X 0,Y 486.184,Z 914.722,A -85,B 0,C 180,E1 17406.065,E2 17406.065} C_VEL
LIN {X 0,Y 484.796,Z 935.025,A -85,B 0,C 180,E1 17405.369,E2 17405.369} C_VEL
LIN {X 0,Y 483.01,Z 954.742,A -85,B 0,C 180,E1 17404.483,E2 17404.483} C_VEL
LIN {X 0,Y 480.96,Z 974.86,A -85,B 0,C 180,E1 17403.358,E2 17403.358} C_VEL
LIN {X 0,Y 478.817,Z 993.209,A -85,B 0,C 180,E1 17402.103,E2 17402.103} C_VEL
LIN {X 0,Y 476.382,Z 1012.475,A -85,B 0,C 180,E1 17400.526,E2 17400.526} C_VEL
LIN {X 0,Y 474.099,Z 1030.262,A -85,B 0,C 180,E1 17398.81,E2 17398.81} C_VEL
LIN {X 0,Y 471.938,Z 1046.567,A -85,B 0,C 180,E1 17396.961,E2 17396.961} C_VEL
LIN {X 0,Y 469.844,Z 1062.981,A -85,B 0,C 180,E1 17394.786,E2 17394.786} C_VEL
LIN {X 0,Y 468.128,Z 1078.244,A -85,B 0,C 180,E1 17392.478,E2 17392.478} C_VEL
LIN {X 0,Y 466.792,Z 1091.277,A -85,B 0,C 180,E1 17390.173,E2 17390.173} C_VEL
LIN {X 0,Y 465.722,Z 1102.833,A -85,B 0,C 180,E1 17387.75,E2 17387.75} C_VEL
LIN {X 0,Y 464.94,Z 1113.014,A -85,B 0,C 180,E1 17385.21,E2 17385.21} C_VEL
LIN {X 0,Y 464.436,Z 1121.425,A -85,B 0,C 180,E1 17382.685,E2 17382.685} C_VEL
LIN {X 0,Y 464.13,Z 1128.065,A -85,B 0,C 180,E1 17380.175,E2 17380.175} C_VEL
LIN {X 0,Y 463.966,Z 1133.411,A -85,B 0,C 180,E1 17377.554,E2 17377.554} C_VEL
LIN {X 0,Y 463.907,Z 1137.022,A -85,B 0,C 180,E1 17375.07,E2 17375.07} C_VEL
LIN {X 0,Y 463.897,Z 1139.219,A -85,B 0,C 180,E1 17372.471,E2 17372.471} C_VEL
LIN {X 0,Y 463.909,Z 1139.989,A -85,B 0,C 180,E1 17369.876,E2 17369.876} C_VEL
LIN {X 0,Y 463.896,Z 1139.135,A -85,B 0,C 180,E1 17367.282,E2 17367.282} C_VEL
LIN {X 0,Y 463.917,Z 1136.658,A -85,B 0,C 180,E1 17364.558,E2 17364.558} C_VEL
LIN {X 0,Y 463.988,Z 1132.941,A -85,B 0,C 180,E1 17362.073,E2 17362.073} C_VEL
LIN {X 0,Y 464.164,Z 1127.372,A -85,B 0,C 180,E1 17359.45,E2 17359.45} C_VEL
LIN {X 0,Y 464.507,Z 1120.148,A -85,B 0,C 180,E1 17356.811,E2 17356.811} C_VEL
LIN {X 0,Y 465.053,Z 1111.5,A -85,B 0,C 180,E1 17354.282,E2 17354.282} C_VEL
LIN {X 0,Y 465.878,Z 1100.939,A -85,B 0,C 180,E1 17351.739,E2 17351.739} C_VEL
LIN {X 0,Y 467.008,Z 1088.998,A -85,B 0,C 180,E1 17349.313,E2 17349.313} C_VEL
LIN {X 0,Y 468.426,Z 1075.679,A -85,B 0,C 180,E1 17347.007,E2 17347.007} C_VEL
LIN {X 0,Y 470.219,Z 1059.935,A -85,B 0,C 180,E1 17344.697,E2 17344.697} C_VEL
LIN {X 0,Y 472.257,Z 1044.05,A -85,B 0,C 180,E1 17342.649,E2 17342.649} C_VEL
LIN {X 0,Y 474.477,Z 1027.383,A -85,B 0,C 180,E1 17340.801,E2 17340.801} C_VEL
LIN {X 0,Y 476.74,Z 1009.857,A -85,B 0,C 180,E1 17339.15,E2 17339.15} C_VEL
LIN {X 0,Y 479.087,Z 990.852,A -85,B 0,C 180,E1 17337.634,E2 17337.634} C_VEL
LIN {X 0,Y 481.256,Z 972.221,A -85,B 0,C 180,E1 17336.387,E2 17336.387} C_VEL
LIN {X 0,Y 483.237,Z 952.576,A -85,B 0,C 180,E1 17335.319,E2 17335.319} C_VEL
LIN {X 0,Y 485.066,Z 931.03,A -85,B 0,C 180,E1 17334.391,E2 17334.391} C_VEL
LIN {X 0,Y 486.481,Z 910.051,A -85,B 0,C 180,E1 17333.706,E2 17333.706} C_VEL
LIN {X 0,Y 487.456,Z 888.25,A -85,B 0,C 180,E1 17333.228,E2 17333.228} C_VEL
LIN {X 0,Y 491.293,Z 704.567,A -85,B 0,C 180,E1 17330.208,E2 17330.208} C_VEL
LIN {X 0,Y 492.952,Z 620.334,A -85,B 0,C 180,E1 17328.808,E2 17328.808} C_VEL
LIN {X 0,Y 486.211,Z 586.575,A -85,B 0,C 180,E1 17327.344,E2 17327.344} C_VEL
LIN {X 0,Y 487.25,Z 575.1,A -85,B 0,C 180,E1 17326.247,E2 17326.247} C_VEL
LIN {X 0,Y 480.532,Z 558.69,A -85,B 0,C 180,E1 17323.606,E2 17323.606} C_VEL
LIN {X 0,Y 474.448,Z 545.292,A -85,B 0,C 180,E1 17321.206,E2 17321.206} C_VEL
LIN {X 0,Y 470.487,Z 537.087,A -85,B 0,C 180,E1 17319.609,E2 17319.609} C_VEL
LIN {X 0,Y 469.924,Z 536.419,A -85,B 0,C 180,E1 17319.434,E2 17319.434} C_VEL
LIN {X 0,Y 469.286,Z 536.543,A -85,B 0,C 180,E1 17319.204,E2 17319.204} C_VEL
LIN {X 0,Y 471.103,Z 541.822,A -85,B 0,C 180,E1 17318.547,E2 17318.547} C_VEL
LIN {X 0,Y 477.005,Z 559.268,A -85,B 0,C 180,E1 17316.6,E2 17316.6} C_VEL
LIN {X 0,Y 475.664,Z 602.889,A -85,B 0,C 180,E1 17312.986,E2 17312.986} C_VEL
LIN {X 0,Y 474.331,Z 642.571,A -85,B 0,C 180,E1 17309.694,E2 17309.694} C_VEL
LIN {X 0,Y 472.701,Z 685.834,A -85,B 0,C 180,E1 17306.102,E2 17306.102} C_VEL
LIN {X 0,Y 471.701,Z 713.996,A -85,B 0,C 180,E1 17303.797,E2 17303.797} C_VEL
LIN {X 0,Y 472.709,Z 723.804,A -85,B 0,C 180,E1 17303.578,E2 17303.578} C_VEL
LIN {X 0,Y 470.617,Z 884.852,A -85,B 0,C 180,E1 17300.92,E2 17300.92} C_VEL
LIN {X 0,Y 470.257,Z 902.284,A -85,B 0,C 180,E1 17300.404,E2 17300.404} C_VEL
LIN {X 0,Y 469.689,Z 919.495,A -85,B 0,C 180,E1 17299.655,E2 17299.655} C_VEL
LIN {X 0,Y 469.024,Z 935.629,A -85,B 0,C 180,E1 17298.714,E2 17298.714} C_VEL
LIN {X 0,Y 468.296,Z 949.94,A -85,B 0,C 180,E1 17297.649,E2 17297.649} C_VEL
LIN {X 0,Y 467.509,Z 964.059,A -85,B 0,C 180,E1 17296.334,E2 17296.334} C_VEL
LIN {X 0,Y 466.726,Z 977.142,A -85,B 0,C 180,E1 17294.833,E2 17294.833} C_VEL
LIN {X 0,Y 466.058,Z 988.263,A -85,B 0,C 180,E1 17293.271,E2 17293.271} C_VEL
LIN {X 0,Y 465.484,Z 998.372,A -85,B 0,C 180,E1 17291.523,E2 17291.523} C_VEL
LIN {X 0,Y 465.029,Z 1006.974,A -85,B 0,C 180,E1 17289.655,E2 17289.655} C_VEL
LIN {X 0,Y 464.703,Z 1014.119,A -85,B 0,C 180,E1 17287.666,E2 17287.666} C_VEL
LIN {X 0,Y 464.524,Z 1019.744,A -85,B 0,C 180,E1 17285.559,E2 17285.559} C_VEL
LIN {X 0,Y 464.438,Z 1023.459,A -85,B 0,C 180,E1 17283.456,E2 17283.456} C_VEL
LIN {X 0,Y 464.42,Z 1025.564,A -85,B 0,C 180,E1 17281.234,E2 17281.234} C_VEL
LIN {X 0,Y 464.446,Z 1025.898,A -85,B 0,C 180,E1 17279.137,E2 17279.137} C_VEL
LIN {X 0,Y 464.486,Z 1024.569,A -85,B 0,C 180,E1 17277.039,E2 17277.039} C_VEL
LIN {X 0,Y 464.587,Z 1021.543,A -85,B 0,C 180,E1 17274.938,E2 17274.938} C_VEL
LIN {X 0,Y 464.796,Z 1016.747,A -85,B 0,C 180,E1 17272.833,E2 17272.833} C_VEL
LIN {X 0,Y 465.117,Z 1010.413,A -85,B 0,C 180,E1 17270.847,E2 17270.847} C_VEL
LIN {X 0,Y 465.55,Z 1002.471,A -85,B 0,C 180,E1 17268.962,E2 17268.962} C_VEL
LIN {X 0,Y 466.128,Z 992.571,A -85,B 0,C 180,E1 17267.11,E2 17267.11} C_VEL
LIN {X 0,Y 466.785,Z 981.748,A -85,B 0,C 180,E1 17265.486,E2 17265.486} C_VEL
LIN {X 0,Y 467.51,Z 969.288,A -85,B 0,C 180,E1 17263.985,E2 17263.985} C_VEL
LIN {X 0,Y 468.219,Z 955.643,A -85,B 0,C 180,E1 17262.66,E2 17262.66} C_VEL
LIN {X 0,Y 468.857,Z 941.218,A -85,B 0,C 180,E1 17261.538,E2 17261.538} C_VEL
LIN {X 0,Y 469.428,Z 925.65,A -85,B 0,C 180,E1 17260.594,E2 17260.594} C_VEL
LIN {X 0,Y 469.87,Z 908.924,A -85,B 0,C 180,E1 17259.839,E2 17259.839} C_VEL
LIN {X 0,Y 470.136,Z 891.423,A -85,B 0,C 180,E1 17259.295,E2 17259.295} C_VEL
LIN {X 0,Y 470.296,Z 865.465,A -85,B 0,C 180,E1 17258.837,E2 17258.837} C_VEL
LIN {X 0,Y 471.815,Z 747.5,A -85,B 0,C 180,E1 17256.906,E2 17256.906} C_VEL
LIN {X 0,Y 472.258,Z 721.669,A -85,B 0,C 180,E1 17256.443,E2 17256.443} C_VEL
LIN {X 0,Y 473.338,Z 680.015,A -85,B 0,C 180,E1 17253.193,E2 17253.193} C_VEL
LIN {X 0,Y 473.876,Z 642.333,A -85,B 0,C 180,E1 17250.352,E2 17250.352} C_VEL
LIN {X 0,Y 473.89,Z 604.95,A -85,B 0,C 180,E1 17247.666,E2 17247.666} C_VEL
LIN {X 0,Y 473.422,Z 565.956,A -85,B 0,C 180,E1 17245.03,E2 17245.03} C_VEL
LIN {X 0,Y 472.804,Z 549.497,A -85,B 0,C 180,E1 17243.957,E2 17243.957} C_VEL
LIN {X 0,Y 470.123,Z 538.713,A -85,B 0,C 180,E1 17243.1,E2 17243.1} C_VEL
LIN {X 0,Y 468.936,Z 534.774,A -85,B 0,C 180,E1 17242.712,E2 17242.712} C_VEL
LIN {X 0,Y 469.585,Z 534.527,A -85,B 0,C 180,E1 17242.486,E2 17242.486} C_VEL
LIN {X 0,Y 476.437,Z 548.747,A -85,B 0,C 180,E1 17239.84,E2 17239.84} C_VEL
LIN {X 0,Y 489.091,Z 567.173,A -85,B 0,C 180,E1 17237.853,E2 17237.853} C_VEL
LIN {X 0,Y 497.749,Z 580.773,A -85,B 0,C 180,E1 17236.579,E2 17236.579} C_VEL
LIN {X 0,Y 492.775,Z 789.544,A -85,B 0,C 180,E1 17232.986,E2 17232.986} C_VEL
LIN {X 0,Y 490.459,Z 893.731,A -85,B 0,C 180,E1 17231.223,E2 17231.223} C_VEL
LIN {X 0,Y 489.28,Z 916.306,A -85,B 0,C 180,E1 17230.65,E2 17230.65} C_VEL
LIN {X 0,Y 487.853,Z 938.393,A -85,B 0,C 180,E1 17229.904,E2 17229.904} C_VEL
LIN {X 0,Y 486.024,Z 959.941,A -85,B 0,C 180,E1 17228.957,E2 17228.957} C_VEL
LIN {X 0,Y 483.967,Z 981.924,A -85,B 0,C 180,E1 17227.775,E2 17227.775} C_VEL
LIN {X 0,Y 481.853,Z 1001.888,A -85,B 0,C 180,E1 17226.477,E2 17226.477} C_VEL
LIN {X 0,Y 479.332,Z 1023.647,A -85,B 0,C 180,E1 17224.805,E2 17224.805} C_VEL
LIN {X 0,Y 477.2,Z 1041.233,A -85,B 0,C 180,E1 17223.224,E2 17223.224} C_VEL
LIN {X 0,Y 474.655,Z 1059.888,A -85,B 0,C 180,E1 17221.212,E2 17221.212} C_VEL
LIN {X 0,Y 472.396,Z 1076.667,A -85,B 0,C 180,E1 17219.131,E2 17219.131} C_VEL
LIN {X 0,Y 470.359,Z 1091.978,A -85,B 0,C 180,E1 17216.922,E2 17216.922} C_VEL
LIN {X 0,Y 468.519,Z 1106.939,A -85,B 0,C 180,E1 17214.457,E2 17214.457} C_VEL
LIN {X 0,Y 467.056,Z 1119.713,A -85,B 0,C 180,E1 17212.002,E2 17212.002} C_VEL
LIN {X 0,Y 465.816,Z 1132.322,A -85,B 0,C 180,E1 17209.172,E2 17209.172} C_VEL
LIN {X 0,Y 465.033,Z 1141.98,A -85,B 0,C 180,E1 17206.616,E2 17206.616} C_VEL
LIN {X 0,Y 464.462,Z 1150.7,A -85,B 0,C 180,E1 17203.825,E2 17203.825} C_VEL
LIN {X 0,Y 464.155,Z 1157.772,A -85,B 0,C 180,E1 17201.053,E2 17201.053} C_VEL
LIN {X 0,Y 463.989,Z 1163.048,A -85,B 0,C 180,E1 17198.301,E2 17198.301} C_VEL
LIN {X 0,Y 463.91,Z 1166.915,A -85,B 0,C 180,E1 17195.566,E2 17195.566} C_VEL
LIN {X 0,Y 463.894,Z 1169.121,A -85,B 0,C 180,E1 17192.842,E2 17192.842} C_VEL
LIN {X 0,Y 463.895,Z 1169.962,A -85,B 0,C 180,E1 17190.247,E2 17190.247} C_VEL
LIN {X 0,Y 463.91,Z 1169.325,A -85,B 0,C 180,E1 17187.529,E2 17187.529} C_VEL
LIN {X 0,Y 463.915,Z 1167.5,A -85,B 0,C 180,E1 17185.054,E2 17185.054} C_VEL
LIN {X 0,Y 463.972,Z 1163.874,A -85,B 0,C 180,E1 17182.197,E2 17182.197} C_VEL
LIN {X 0,Y 464.079,Z 1159.319,A -85,B 0,C 180,E1 17179.699,E2 17179.699} C_VEL
LIN {X 0,Y 464.361,Z 1152.818,A -85,B 0,C 180,E1 17176.933,E2 17176.933} C_VEL
LIN {X 0,Y 464.837,Z 1144.934,A -85,B 0,C 180,E1 17174.275,E2 17174.275} C_VEL
LIN {X 0,Y 465.656,Z 1134.385,A -85,B 0,C 180,E1 17171.341,E2 17171.341} C_VEL
LIN {X 0,Y 466.723,Z 1123.234,A -85,B 0,C 180,E1 17168.731,E2 17168.731} C_VEL
LIN {X 0,Y 468.094,Z 1110.446,A -85,B 0,C 180,E1 17166.19,E2 17166.19} C_VEL
LIN {X 0,Y 469.843,Z 1096.204,A -85,B 0,C 180,E1 17163.728,E2 17163.728} C_VEL
LIN {X 0,Y 471.807,Z 1080.927,A -85,B 0,C 180,E1 17161.462,E2 17161.462} C_VEL
LIN {X 0,Y 474.193,Z 1063.218,A -85,B 0,C 180,E1 17159.178,E2 17159.178} C_VEL
LIN {X 0,Y 476.542,Z 1046.215,A -85,B 0,C 180,E1 17157.283,E2 17157.283} C_VEL
LIN {X 0,Y 478.807,Z 1028.081,A -85,B 0,C 180,E1 17155.572,E2 17155.572} C_VEL
LIN {X 0,Y 481.042,Z 1009.108,A -85,B 0,C 180,E1 17154.042,E2 17154.042} C_VEL
LIN {X 0,Y 483.362,Z 987.834,A -85,B 0,C 180,E1 17152.591,E2 17152.591} C_VEL
LIN {X 0,Y 485.442,Z 966.872,A -85,B 0,C 180,E1 17151.385,E2 17151.385} C_VEL
LIN {X 0,Y 487.31,Z 944.544,A -85,B 0,C 180,E1 17150.349,E2 17150.349} C_VEL
LIN {X 0,Y 488.982,Z 921.618,A -85,B 0,C 180,E1 17149.508,E2 17149.508} C_VEL
LIN {X 0,Y 490.116,Z 900.839,A -85,B 0,C 180,E1 17148.941,E2 17148.941} C_VEL
LIN {X 0,Y 491.009,Z 874.606,A -85,B 0,C 180,E1 17148.433,E2 17148.433} C_VEL
LIN {X 0,Y 495.086,Z 687.966,A -85,B 0,C 180,E1 17145.282,E2 17145.282} C_VEL
LIN {X 0,Y 497.716,Z 578.827,A -85,B 0,C 180,E1 17143.376,E2 17143.376} C_VEL
LIN {X 0,Y 483.391,Z 557.194,A -85,B 0,C 180,E1 17141.247,E2 17141.247} C_VEL
LIN {X 0,Y 476.472,Z 547.214,A -85,B 0,C 180,E1 17140.107,E2 17140.107} C_VEL
LIN {X 0,Y 471.219,Z 537.458,A -85,B 0,C 180,E1 17138.44,E2 17138.44} C_VEL
LIN {X 0,Y 469.148,Z 533.575,A -85,B 0,C 180,E1 17137.75,E2 17137.75} C_VEL
LIN {X 0,Y 466.927,Z 529.39,A -85,B 0,C 180,E1 17136.991,E2 17136.991} C_VEL
LIN {X 0,Y 465.221,Z 526.22,A -85,B 0,C 180,E1 17136.383,E2 17136.383} C_VEL
LIN {X 0,Y 465.019,Z 525.223,A -85,B 0,C 180,E1 17136.095,E2 17136.095} C_VEL
LIN {X 0,Y 464.996,Z 525.088,A -85,B 0,C 180,E1 17132.371,E2 17132.371} C_VEL
LIN {X 0,Y 465.013,Z 525.102,A -85,B 0,C 180,E1 17128.685,E2 17128.685} C_VEL
LIN {X 0,Y 465.004,Z 525.124,A -85,B 0,C 180,E1 17124.925,E2 17124.925} C_VEL
LIN {X 0,Y 465.008,Z 525.083,A -85,B 0,C 180,E1 17121.176,E2 17121.176} C_VEL
LIN {X 0,Y 465.001,Z 525.114,A -85,B 0,C 180,E1 17117.519,E2 17117.519} C_VEL
LIN {X 0,Y 465.011,Z 525.097,A -85,B 0,C 180,E1 17113.808,E2 17113.808} C_VEL
LIN {X 0,Y 464.997,Z 525.098,A -85,B 0,C 180,E1 17110.155,E2 17110.155} C_VEL
LIN {X 0,Y 465.011,Z 525.108,A -85,B 0,C 180,E1 17106.419,E2 17106.419} C_VEL
LIN {X 0,Y 465.002,Z 525.114,A -85,B 0,C 180,E1 17102.711,E2 17102.711} C_VEL
LIN {X 0,Y 465.011,Z 525.117,A -85,B 0,C 180,E1 17099.014,E2 17099.014} C_VEL
LIN {X 0,Y 464.998,Z 525.122,A -85,B 0,C 180,E1 17095.313,E2 17095.313} C_VEL
LIN {X 0,Y 465.011,Z 525.117,A -85,B 0,C 180,E1 17091.717,E2 17091.717} C_VEL
LIN {X 0,Y 465.003,Z 525.082,A -85,B 0,C 180,E1 17088.057,E2 17088.057} C_VEL
LIN {X 0,Y 465.001,Z 525.124,A -85,B 0,C 180,E1 17084.408,E2 17084.408} C_VEL
LIN {X 0,Y 464.992,Z 525.082,A -85,B 0,C 180,E1 17080.662,E2 17080.662} C_VEL
LIN {X 0,Y 465.013,Z 525.119,A -85,B 0,C 180,E1 17076.967,E2 17076.967} C_VEL
LIN {X 0,Y 465.007,Z 525.098,A -85,B 0,C 180,E1 17073.295,E2 17073.295} C_VEL
LIN {X 0,Y 464.989,Z 525.092,A -85,B 0,C 180,E1 17069.79,E2 17069.79} C_VEL
LIN {X 0,Y 465.003,Z 525.121,A -85,B 0,C 180,E1 17066.098,E2 17066.098} C_VEL
LIN {X 0,Y 465.011,Z 525.114,A -85,B 0,C 180,E1 17062.363,E2 17062.363} C_VEL
LIN {X 0,Y 465.028,Z 525.37,A -85,B 0,C 180,E1 17061.393,E2 17061.393} C_VEL
LIN {X 0,Y 466.633,Z 529.015,A -85,B 0,C 180,E1 17060.671,E2 17060.671} C_VEL
LIN {X 0,Y 467.791,Z 531.024,A -85,B 0,C 180,E1 17060.276,E2 17060.276} C_VEL
LIN {X 0,Y 474.592,Z 544.027,A -85,B 0,C 180,E1 17057.936,E2 17057.936} C_VEL
LIN {X 0,Y 482.58,Z 560.449,A -85,B 0,C 180,E1 17055.289,E2 17055.289} C_VEL
LIN {X 0,Y 489.098,Z 575.025,A -85,B 0,C 180,E1 17053.176,E2 17053.176} C_VEL
LIN {X 0,Y 488.256,Z 586.705,A -85,B 0,C 180,E1 17052.288,E2 17052.288} C_VEL
LIN {X 0,Y 493.172,Z 617.609,A -85,B 0,C 180,E1 17051.127,E2 17051.127} C_VEL
LIN {X 0,Y 491.329,Z 703.643,A -85,B 0,C 180,E1 17049.712,E2 17049.712} C_VEL
LIN {X 0,Y 490.427,Z 711.347,A -85,B 0,C 180,E1 17049.667,E2 17049.667} C_VEL
LIN {X 0,Y 485.391,Z 731.943,A -85,B 0,C 180,E1 17049.831,E2 17049.831} C_VEL
LIN {X 0,Y 484.699,Z 738.554,A -85,B 0,C 180,E1 17049.783,E2 17049.783} C_VEL
LIN {X 0,Y 481.218,Z 895.349,A -85,B 0,C 180,E1 17047.181,E2 17047.181} C_VEL
LIN {X 0,Y 480.045,Z 916.45,A -85,B 0,C 180,E1 17046.646,E2 17046.646} C_VEL
LIN {X 0,Y 478.597,Z 936.401,A -85,B 0,C 180,E1 17045.948,E2 17045.948} C_VEL
LIN {X 0,Y 476.608,Z 956.669,A -85,B 0,C 180,E1 17045.013,E2 17045.013} C_VEL
LIN {X 0,Y 474.302,Z 977.338,A -85,B 0,C 180,E1 17043.816,E2 17043.816} C_VEL
LIN {X 0,Y 471.95,Z 996.312,A -85,B 0,C 180,E1 17042.484,E2 17042.484} C_VEL
LIN {X 0,Y 469.362,Z 1015.058,A -85,B 0,C 180,E1 17040.89,E2 17040.89} C_VEL
LIN {X 0,Y 466.74,Z 1033.472,A -85,B 0,C 180,E1 17039.034,E2 17039.034} C_VEL
LIN {X 0,Y 464.327,Z 1050.451,A -85,B 0,C 180,E1 17037.024,E2 17037.024} C_VEL
LIN {X 0,Y 462.244,Z 1065.428,A -85,B 0,C 180,E1 17034.948,E2 17034.948} C_VEL
LIN {X 0,Y 460.435,Z 1079.109,A -85,B 0,C 180,E1 17032.739,E2 17032.739} C_VEL
LIN {X 0,Y 458.782,Z 1093.824,A -85,B 0,C 180,E1 17030.009,E2 17030.009} C_VEL
LIN {X 0,Y 457.71,Z 1105.073,A -85,B 0,C 180,E1 17027.545,E2 17027.545} C_VEL
LIN {X 0,Y 456.913,Z 1114.85,A -85,B 0,C 180,E1 17024.964,E2 17024.964} C_VEL
LIN {X 0,Y 456.376,Z 1123.195,A -85,B 0,C 180,E1 17022.27,E2 17022.27} C_VEL
LIN {X 0,Y 456.096,Z 1129.538,A -85,B 0,C 180,E1 17019.718,E2 17019.718} C_VEL
LIN {X 0,Y 455.958,Z 1134.24,A -85,B 0,C 180,E1 17017.18,E2 17017.18} C_VEL
LIN {X 0,Y 455.916,Z 1137.79,A -85,B 0,C 180,E1 17014.402,E2 17014.402} C_VEL
LIN {X 0,Y 455.9,Z 1139.558,A -85,B 0,C 180,E1 17011.885,E2 17011.885} C_VEL
LIN {X 0,Y 455.896,Z 1139.877,A -85,B 0,C 180,E1 17009.246,E2 17009.246} C_VEL
LIN {X 0,Y 455.909,Z 1138.778,A -85,B 0,C 180,E1 17006.605,E2 17006.605} C_VEL
LIN {X 0,Y 455.94,Z 1136.018,A -85,B 0,C 180,E1 17003.958,E2 17003.958} C_VEL
LIN {X 0,Y 456.045,Z 1131.498,A -85,B 0,C 180,E1 17001.172,E2 17001.172} C_VEL
LIN {X 0,Y 456.278,Z 1125.549,A -85,B 0,C 180,E1 16998.497,E2 16998.497} C_VEL
LIN {X 0,Y 456.695,Z 1118.012,A -85,B 0,C 180,E1 16995.902,E2 16995.902} C_VEL
LIN {X 0,Y 457.397,Z 1108.513,A -85,B 0,C 180,E1 16993.228,E2 16993.228} C_VEL
LIN {X 0,Y 458.37,Z 1098.059,A -85,B 0,C 180,E1 16990.769,E2 16990.769} C_VEL
LIN {X 0,Y 459.691,Z 1085.485,A -85,B 0,C 180,E1 16988.299,E2 16988.299} C_VEL
LIN {X 0,Y 461.51,Z 1070.813,A -85,B 0,C 180,E1 16985.797,E2 16985.797} C_VEL
LIN {X 0,Y 463.54,Z 1055.98,A -85,B 0,C 180,E1 16983.619,E2 16983.619} C_VEL
LIN {X 0,Y 465.756,Z 1040.462,A -85,B 0,C 180,E1 16981.663,E2 16981.663} C_VEL
LIN {X 0,Y 468.181,Z 1023.398,A -85,B 0,C 180,E1 16979.822,E2 16979.822} C_VEL
LIN {X 0,Y 470.752,Z 1005.121,A -85,B 0,C 180,E1 16978.143,E2 16978.143} C_VEL
LIN {X 0,Y 473.111,Z 987.016,A -85,B 0,C 180,E1 16976.741,E2 16976.741} C_VEL
LIN {X 0,Y 475.473,Z 967.255,A -85,B 0,C 180,E1 16975.478,E2 16975.478} C_VEL
LIN {X 0,Y 477.574,Z 947.476,A -85,B 0,C 180,E1 16974.443,E2 16974.443} C_VEL
LIN {X 0,Y 479.318,Z 926.725,A -85,B 0,C 180,E1 16973.596,E2 16973.596} C_VEL
LIN {X 0,Y 480.736,Z 905.247,A -85,B 0,C 180,E1 16972.955,E2 16972.955} C_VEL
LIN {X 0,Y 481.655,Z 882.65,A -85,B 0,C 180,E1 16972.496,E2 16972.496} C_VEL
LIN {X 0,Y 486.269,Z 667.179,A -85,B 0,C 180,E1 16968.954,E2 16968.954} C_VEL
LIN {X 0,Y 487.127,Z 621.94,A -85,B 0,C 180,E1 16968.178,E2 16968.178} C_VEL
LIN {X 0,Y 480.032,Z 585.992,A -85,B 0,C 180,E1 16966.578,E2 16966.578} C_VEL
LIN {X 0,Y 480.65,Z 578.713,A -85,B 0,C 180,E1 16965.863,E2 16965.863} C_VEL
LIN {X 0,Y 473.711,Z 561.922,A -85,B 0,C 180,E1 16963.088,E2 16963.088} C_VEL
LIN {X 0,Y 467.257,Z 547.365,A -85,B 0,C 180,E1 16960.419,E2 16960.419} C_VEL
LIN {X 0,Y 464.915,Z 542.879,A -85,B 0,C 180,E1 16959.498,E2 16959.498} C_VEL
LIN {X 0,Y 463.495,Z 542.767,A -85,B 0,C 180,E1 16959.203,E2 16959.203} C_VEL
LIN {X 0,Y 463.616,Z 543.79,A -85,B 0,C 180,E1 16958.97,E2 16958.97} C_VEL
LIN {X 0,Y 469.815,Z 562.175,A -85,B 0,C 180,E1 16956.881,E2 16956.881} C_VEL
LIN {X 0,Y 468.36,Z 606.433,A -85,B 0,C 180,E1 16953.191,E2 16953.191} C_VEL
LIN {X 0,Y 466.95,Z 646.323,A -85,B 0,C 180,E1 16949.864,E2 16949.864} C_VEL
LIN {X 0,Y 465.252,Z 689.256,A -85,B 0,C 180,E1 16946.277,E2 16946.277} C_VEL
LIN {X 0,Y 464.325,Z 715.078,A -85,B 0,C 180,E1 16944.158,E2 16944.158} C_VEL
LIN {X 0,Y 465.282,Z 724.719,A -85,B 0,C 180,E1 16943.932,E2 16943.932} C_VEL
LIN {X 0,Y 463.034,Z 886.113,A -85,B 0,C 180,E1 16941.213,E2 16941.213} C_VEL
LIN {X 0,Y 462.663,Z 903.559,A -85,B 0,C 180,E1 16940.685,E2 16940.685} C_VEL
LIN {X 0,Y 462.079,Z 920.724,A -85,B 0,C 180,E1 16939.926,E2 16939.926} C_VEL
LIN {X 0,Y 461.389,Z 936.88,A -85,B 0,C 180,E1 16938.969,E2 16938.969} C_VEL
LIN {X 0,Y 460.586,Z 951.934,A -85,B 0,C 180,E1 16937.824,E2 16937.824} C_VEL
LIN {X 0,Y 459.746,Z 966.356,A -85,B 0,C 180,E1 16936.445,E2 16936.445} C_VEL
LIN {X 0,Y 458.932,Z 979.472,A -85,B 0,C 180,E1 16934.897,E2 16934.897} C_VEL
LIN {X 0,Y 458.213,Z 990.817,A -85,B 0,C 180,E1 16933.246,E2 16933.246} C_VEL
LIN {X 0,Y 457.616,Z 1000.67,A -85,B 0,C 180,E1 16931.469,E2 16931.469} C_VEL
LIN {X 0,Y 457.156,Z 1009.128,A -85,B 0,C 180,E1 16929.569,E2 16929.569} C_VEL
LIN {X 0,Y 456.832,Z 1016.144,A -85,B 0,C 180,E1 16927.546,E2 16927.546} C_VEL
LIN {X 0,Y 456.649,Z 1021.301,A -85,B 0,C 180,E1 16925.529,E2 16925.529} C_VEL
LIN {X 0,Y 456.56,Z 1024.971,A -85,B 0,C 180,E1 16923.39,E2 16923.39} C_VEL
LIN {X 0,Y 456.549,Z 1027.044,A -85,B 0,C 180,E1 16921.13,E2 16921.13} C_VEL
LIN {X 0,Y 456.581,Z 1027.309,A -85,B 0,C 180,E1 16918.997,E2 16918.997} C_VEL
LIN {X 0,Y 456.628,Z 1025.858,A -85,B 0,C 180,E1 16916.85,E2 16916.85} C_VEL
LIN {X 0,Y 456.767,Z 1022.527,A -85,B 0,C 180,E1 16914.599,E2 16914.599} C_VEL
LIN {X 0,Y 456.999,Z 1017.85,A -85,B 0,C 180,E1 16912.584,E2 16912.584} C_VEL
LIN {X 0,Y 457.355,Z 1011.313,A -85,B 0,C 180,E1 16910.563,E2 16910.563} C_VEL
LIN {X 0,Y 457.826,Z 1003.289,A -85,B 0,C 180,E1 16908.665,E2 16908.665} C_VEL
LIN {X 0,Y 458.419,Z 993.826,A -85,B 0,C 180,E1 16906.89,E2 16906.89} C_VEL
LIN {X 0,Y 459.119,Z 982.781,A -85,B 0,C 180,E1 16905.226,E2 16905.226} C_VEL
LIN {X 0,Y 459.871,Z 970.241,A -85,B 0,C 180,E1 16903.712,E2 16903.712} C_VEL
LIN {X 0,Y 460.623,Z 956.273,A -85,B 0,C 180,E1 16902.35,E2 16902.35} C_VEL
LIN {X 0,Y 461.281,Z 941.758,A -85,B 0,C 180,E1 16901.224,E2 16901.224} C_VEL
LIN {X 0,Y 461.853,Z 925.686,A -85,B 0,C 180,E1 16900.262,E2 16900.262} C_VEL
LIN {X 0,Y 462.293,Z 908.511,A -85,B 0,C 180,E1 16899.502,E2 16899.502} C_VEL
LIN {X 0,Y 462.518,Z 891.268,A -85,B 0,C 180,E1 16898.987,E2 16898.987} C_VEL
LIN {X 0,Y 464.356,Z 749.258,A -85,B 0,C 180,E1 16896.572,E2 16896.572} C_VEL
LIN {X 0,Y 464.898,Z 723.459,A -85,B 0,C 180,E1 16896.084,E2 16896.084} C_VEL
LIN {X 0,Y 465.851,Z 693.896,A -85,B 0,C 180,E1 16893.76,E2 16893.76} C_VEL
LIN {X 0,Y 466.591,Z 654.521,A -85,B 0,C 180,E1 16890.753,E2 16890.753} C_VEL
LIN {X 0,Y 466.828,Z 615.686,A -85,B 0,C 180,E1 16887.916,E2 16887.916} C_VEL
LIN {X 0,Y 466.477,Z 579.224,A -85,B 0,C 180,E1 16885.389,E2 16885.389} C_VEL
LIN {X 0,Y 465.851,Z 552.2,A -85,B 0,C 180,E1 16883.598,E2 16883.598} C_VEL
LIN {X 0,Y 463.459,Z 542.191,A -85,B 0,C 180,E1 16882.757,E2 16882.757} C_VEL
LIN {X 0,Y 463.889,Z 541.474,A -85,B 0,C 180,E1 16882.53,E2 16882.53} C_VEL
LIN {X 0,Y 464.654,Z 541.766,A -85,B 0,C 180,E1 16882.361,E2 16882.361} C_VEL
LIN {X 0,Y 468.702,Z 549.787,A -85,B 0,C 180,E1 16880.844,E2 16880.844} C_VEL
LIN {X 0,Y 481.413,Z 567.999,A -85,B 0,C 180,E1 16878.764,E2 16878.764} C_VEL
LIN {X 0,Y 491.904,Z 584.298,A -85,B 0,C 180,E1 16877.167,E2 16877.167} C_VEL
LIN {X 0,Y 486.359,Z 798.261,A -85,B 0,C 180,E1 16873.431,E2 16873.431} C_VEL
LIN {X 0,Y 484.022,Z 893.685,A -85,B 0,C 180,E1 16871.787,E2 16871.787} C_VEL
LIN {X 0,Y 482.754,Z 916.44,A -85,B 0,C 180,E1 16871.201,E2 16871.201} C_VEL
LIN {X 0,Y 481.172,Z 939.186,A -85,B 0,C 180,E1 16870.416,E2 16870.416} C_VEL
LIN {X 0,Y 479.248,Z 960.895,A -85,B 0,C 180,E1 16869.449,E2 16869.449} C_VEL
LIN {X 0,Y 476.937,Z 984.01,A -85,B 0,C 180,E1 16868.173,E2 16868.173} C_VEL
LIN {X 0,Y 474.766,Z 1003.372,A -85,B 0,C 180,E1 16866.885,E2 16866.885} C_VEL
LIN {X 0,Y 472.226,Z 1023.937,A -85,B 0,C 180,E1 16865.269,E2 16865.269} C_VEL
LIN {X 0,Y 469.822,Z 1042.745,A -85,B 0,C 180,E1 16863.551,E2 16863.551} C_VEL
LIN {X 0,Y 467.379,Z 1060.883,A -85,B 0,C 180,E1 16861.61,E2 16861.61} C_VEL
LIN {X 0,Y 465.407,Z 1074.639,A -85,B 0,C 180,E1 16859.896,E2 16859.896} C_VEL
LIN {X 0,Y 463.059,Z 1091.131,A -85,B 0,C 180,E1 16857.521,E2 16857.521} C_VEL
LIN {X 0,Y 461.137,Z 1105.501,A -85,B 0,C 180,E1 16855.149,E2 16855.149} C_VEL
LIN {X 0,Y 459.514,Z 1118.441,A -85,B 0,C 180,E1 16852.652,E2 16852.652} C_VEL
LIN {X 0,Y 458.24,Z 1130.252,A -85,B 0,C 180,E1 16850.033,E2 16850.033} C_VEL
LIN {X 0,Y 457.304,Z 1140.144,A -85,B 0,C 180,E1 16847.43,E2 16847.43} C_VEL
LIN {X 0,Y 456.621,Z 1149.32,A -85,B 0,C 180,E1 16844.572,E2 16844.572} C_VEL
LIN {X 0,Y 456.238,Z 1156.258,A -85,B 0,C 180,E1 16841.888,E2 16841.888} C_VEL
LIN {X 0,Y 456.026,Z 1162.222,A -85,B 0,C 180,E1 16838.956,E2 16838.956} C_VEL
LIN {X 0,Y 455.932,Z 1166.119,A -85,B 0,C 180,E1 16836.295,E2 16836.295} C_VEL
LIN {X 0,Y 455.888,Z 1168.849,A -85,B 0,C 180,E1 16833.395,E2 16833.395} C_VEL
LIN {X 0,Y 455.888,Z 1169.849,A -85,B 0,C 180,E1 16830.88,E2 16830.88} C_VEL
LIN {X 0,Y 455.906,Z 1169.658,A -85,B 0,C 180,E1 16828.115,E2 16828.115} C_VEL
LIN {X 0,Y 455.91,Z 1167.841,A -85,B 0,C 180,E1 16825.346,E2 16825.346} C_VEL
LIN {X 0,Y 455.943,Z 1164.681,A -85,B 0,C 180,E1 16822.566,E2 16822.566} C_VEL
LIN {X 0,Y 456.068,Z 1159.987,A -85,B 0,C 180,E1 16819.851,E2 16819.851} C_VEL
LIN {X 0,Y 456.334,Z 1154.133,A -85,B 0,C 180,E1 16817.215,E2 16817.215} C_VEL
LIN {X 0,Y 456.846,Z 1146.079,A -85,B 0,C 180,E1 16814.361,E2 16814.361} C_VEL
LIN {X 0,Y 457.61,Z 1136.925,A -85,B 0,C 180,E1 16811.661,E2 16811.661} C_VEL
LIN {X 0,Y 458.702,Z 1125.718,A -85,B 0,C 180,E1 16808.921,E2 16808.921} C_VEL
LIN {X 0,Y 460.151,Z 1113.246,A -85,B 0,C 180,E1 16806.298,E2 16806.298} C_VEL
LIN {X 0,Y 461.936,Z 1099.337,A -85,B 0,C 180,E1 16803.797,E2 16803.797} C_VEL
LIN {X 0,Y 464.175,Z 1083.178,A -85,B 0,C 180,E1 16801.291,E2 16801.291} C_VEL
LIN {X 0,Y 466.611,Z 1066.529,A -85,B 0,C 180,E1 16799.051,E2 16799.051} C_VEL
LIN {X 0,Y 468.882,Z 1049.625,A -85,B 0,C 180,E1 16797.158,E2 16797.158} C_VEL
LIN {X 0,Y 471.403,Z 1030.631,A -85,B 0,C 180,E1 16795.308,E2 16795.308} C_VEL
LIN {X 0,Y 473.757,Z 1011.547,A -85,B 0,C 180,E1 16793.726,E2 16793.726} C_VEL
LIN {X 0,Y 476.311,Z 989.9,A -85,B 0,C 180,E1 16792.196,E2 16792.196} C_VEL
LIN {X 0,Y 478.302,Z 970.999,A -85,B 0,C 180,E1 16791.076,E2 16791.076} C_VEL
LIN {X 0,Y 480.396,Z 948.014,A -85,B 0,C 180,E1 16789.952,E2 16789.952} C_VEL
LIN {X 0,Y 482.114,Z 926.066,A -85,B 0,C 180,E1 16789.102,E2 16789.102} C_VEL
LIN {X 0,Y 483.524,Z 903.196,A -85,B 0,C 180,E1 16788.438,E2 16788.438} C_VEL
LIN {X 0,Y 484.501,Z 880.084,A -85,B 0,C 180,E1 16787.956,E2 16787.956} C_VEL
LIN {X 0,Y 489.17,Z 686.249,A -85,B 0,C 180,E1 16784.627,E2 16784.627} C_VEL
LIN {X 0,Y 491.841,Z 582.418,A -85,B 0,C 180,E1 16782.786,E2 16782.786} C_VEL
LIN {X 0,Y 478.886,Z 562.772,A -85,B 0,C 180,E1 16780.806,E2 16780.806} C_VEL
LIN {X 0,Y 468.804,Z 548.443,A -85,B 0,C 180,E1 16779.146,E2 16779.146} C_VEL
LIN {X 0,Y 461.947,Z 535.525,A -85,B 0,C 180,E1 16776.837,E2 16776.837} C_VEL
LIN {X 0,Y 459.71,Z 531.309,A -85,B 0,C 180,E1 16776.038,E2 16776.038} C_VEL
LIN {X 0,Y 457.392,Z 527.566,A -85,B 0,C 180,E1 16775.247,E2 16775.247} C_VEL
LIN {X 0,Y 457.099,Z 526.309,A -85,B 0,C 180,E1 16774.966,E2 16774.966} C_VEL
LIN {X 0,Y 457.063,Z 526.082,A -85,B 0,C 180,E1 16771.375,E2 16771.375} C_VEL
LIN {X 0,Y 457.062,Z 526.075,A -85,B 0,C 180,E1 16767.771,E2 16767.771} C_VEL
LIN {X 0,Y 457.065,Z 526.112,A -85,B 0,C 180,E1 16764.009,E2 16764.009} C_VEL
LIN {X 0,Y 457.064,Z 526.082,A -85,B 0,C 180,E1 16760.354,E2 16760.354} C_VEL
LIN {X 0,Y 457.062,Z 526.08,A -85,B 0,C 180,E1 16756.632,E2 16756.632} C_VEL
LIN {X 0,Y 457.065,Z 526.101,A -85,B 0,C 180,E1 16753.021,E2 16753.021} C_VEL
LIN {X 0,Y 457.065,Z 526.067,A -85,B 0,C 180,E1 16749.316,E2 16749.316} C_VEL
LIN {X 0,Y 457.064,Z 526.113,A -85,B 0,C 180,E1 16745.649,E2 16745.649} C_VEL
LIN {X 0,Y 457.065,Z 526.116,A -85,B 0,C 180,E1 16741.88,E2 16741.88} C_VEL
LIN {X 0,Y 457.067,Z 526.112,A -85,B 0,C 180,E1 16738.245,E2 16738.245} C_VEL
LIN {X 0,Y 457.069,Z 526.112,A -85,B 0,C 180,E1 16734.465,E2 16734.465} C_VEL
LIN {X 0,Y 457.062,Z 526.113,A -85,B 0,C 180,E1 16730.811,E2 16730.811} C_VEL
LIN {X 0,Y 457.057,Z 526.066,A -85,B 0,C 180,E1 16727.106,E2 16727.106} C_VEL
LIN {X 0,Y 457.069,Z 526.112,A -85,B 0,C 180,E1 16723.478,E2 16723.478} C_VEL
LIN {X 0,Y 457.068,Z 526.074,A -85,B 0,C 180,E1 16719.779,E2 16719.779} C_VEL
LIN {X 0,Y 457.054,Z 526.095,A -85,B 0,C 180,E1 16716.264,E2 16716.264} C_VEL
LIN {X 0,Y 457.068,Z 526.104,A -85,B 0,C 180,E1 16712.511,E2 16712.511} C_VEL
LIN {X 0,Y 457.067,Z 526.072,A -85,B 0,C 180,E1 16708.771,E2 16708.771} C_VEL
LIN {X 0,Y 457.068,Z 526.083,A -85,B 0,C 180,E1 16705.118,E2 16705.118} C_VEL
LIN {X 0,Y 457.102,Z 526.333,A -85,B 0,C 180,E1 16702.6,E2 16702.6} C_VEL
LIN {X 0,Y 458.513,Z 529.802,A -85,B 0,C 180,E1 16701.893,E2 16701.893} C_VEL
LIN {X 0,Y 459.931,Z 532.149,A -85,B 0,C 180,E1 16701.397,E2 16701.397} C_VEL
LIN {X 0,Y 462.67,Z 537.321,A -85,B 0,C 180,E1 16700.393,E2 16700.393} C_VEL
LIN {X 0,Y 467.264,Z 546.097,A -85,B 0,C 180,E1 16698.771,E2 16698.771} C_VEL
LIN {X 0,Y 473.805,Z 559.302,A -85,B 0,C 180,E1 16696.532,E2 16696.532} C_VEL
LIN {X 0,Y 481.667,Z 576.443,A -85,B 0,C 180,E1 16693.919,E2 16693.919} C_VEL
LIN {X 0,Y 482.686,Z 579.126,A -85,B 0,C 180,E1 16693.554,E2 16693.554} C_VEL
LIN {X 0,Y 482.228,Z 586.417,A -85,B 0,C 180,E1 16693.012,E2 16693.012} C_VEL
LIN {X 0,Y 487.374,Z 619.14,A -85,B 0,C 180,E1 16691.755,E2 16691.755} C_VEL
LIN {X 0,Y 484.699,Z 738.554,A -85,B 0,C 180,E1 16689.783,E2 16689.783} C_VEL
LIN {X 0,Y 483.804,Z 746.259,A -85,B 0,C 180,E1 16689.737,E2 16689.737} C_VEL
LIN {X 0,Y 478.768,Z 766.855,A -85,B 0,C 180,E1 16689.906,E2 16689.906} C_VEL
LIN {X 0,Y 478.079,Z 773.465,A -85,B 0,C 180,E1 16689.858,E2 16689.858} C_VEL
LIN {X 0,Y 475.263,Z 896.191,A -85,B 0,C 180,E1 16687.814,E2 16687.814} C_VEL
LIN {X 0,Y 474.025,Z 917.28,A -85,B 0,C 180,E1 16687.271,E2 16687.271} C_VEL
LIN {X 0,Y 472.407,Z 937.949,A -85,B 0,C 180,E1 16686.532,E2 16686.532} C_VEL
LIN {X 0,Y 470.394,Z 957.449,A -85,B 0,C 180,E1 16685.62,E2 16685.62} C_VEL
LIN {X 0,Y 467.953,Z 977.931,A -85,B 0,C 180,E1 16684.42,E2 16684.42} C_VEL
LIN {X 0,Y 465.432,Z 996.885,A -85,B 0,C 180,E1 16683.069,E2 16683.069} C_VEL
LIN {X 0,Y 462.656,Z 1015.521,A -85,B 0,C 180,E1 16681.461,E2 16681.461} C_VEL
LIN {X 0,Y 459.953,Z 1033.235,A -85,B 0,C 180,E1 16679.657,E2 16679.657} C_VEL
LIN {X 0,Y 457.436,Z 1049.531,A -85,B 0,C 180,E1 16677.718,E2 16677.718} C_VEL
LIN {X 0,Y 455.029,Z 1065.243,A -85,B 0,C 180,E1 16675.511,E2 16675.511} C_VEL
LIN {X 0,Y 452.937,Z 1079.732,A -85,B 0,C 180,E1 16673.137,E2 16673.137} C_VEL
LIN {X 0,Y 451.227,Z 1092.789,A -85,B 0,C 180,E1 16670.63,E2 16670.63} C_VEL
LIN {X 0,Y 449.827,Z 1105.59,A -85,B 0,C 180,E1 16667.729,E2 16667.729} C_VEL
LIN {X 0,Y 449.013,Z 1114.852,A -85,B 0,C 180,E1 16665.234,E2 16665.234} C_VEL
LIN {X 0,Y 448.428,Z 1123.197,A -85,B 0,C 180,E1 16662.491,E2 16662.491} C_VEL
LIN {X 0,Y 448.117,Z 1129.54,A -85,B 0,C 180,E1 16659.893,E2 16659.893} C_VEL
LIN {X 0,Y 447.964,Z 1134.24,A -85,B 0,C 180,E1 16657.309,E2 16657.309} C_VEL
LIN {X 0,Y 447.915,Z 1137.79,A -85,B 0,C 180,E1 16654.481,E2 16654.481} C_VEL
LIN {X 0,Y 447.901,Z 1139.558,A -85,B 0,C 180,E1 16651.919,E2 16651.919} C_VEL
LIN {X 0,Y 447.896,Z 1139.876,A -85,B 0,C 180,E1 16649.233,E2 16649.233} C_VEL
LIN {X 0,Y 447.91,Z 1138.777,A -85,B 0,C 180,E1 16646.545,E2 16646.545} C_VEL
LIN {X 0,Y 447.944,Z 1136.017,A -85,B 0,C 180,E1 16643.849,E2 16643.849} C_VEL
LIN {X 0,Y 448.059,Z 1131.496,A -85,B 0,C 180,E1 16641.013,E2 16641.013} C_VEL
LIN {X 0,Y 448.318,Z 1125.472,A -85,B 0,C 180,E1 16638.26,E2 16638.26} C_VEL
LIN {X 0,Y 448.762,Z 1118.114,A -85,B 0,C 180,E1 16635.681,E2 16635.681} C_VEL
LIN {X 0,Y 449.539,Z 1108.514,A -85,B 0,C 180,E1 16632.927,E2 16632.927} C_VEL
LIN {X 0,Y 450.672,Z 1097.512,A -85,B 0,C 180,E1 16630.292,E2 16630.292} C_VEL
LIN {X 0,Y 452.194,Z 1085.268,A -85,B 0,C 180,E1 16627.784,E2 16627.784} C_VEL
LIN {X 0,Y 454.078,Z 1071.661,A -85,B 0,C 180,E1 16625.407,E2 16625.407} C_VEL
LIN {X 0,Y 456.31,Z 1056.765,A -85,B 0,C 180,E1 16623.167,E2 16623.167} C_VEL
LIN {X 0,Y 458.796,Z 1040.747,A -85,B 0,C 180,E1 16621.108,E2 16621.108} C_VEL
LIN {X 0,Y 461.426,Z 1023.676,A -85,B 0,C 180,E1 16619.244,E2 16619.244} C_VEL
LIN {X 0,Y 464.251,Z 1004.849,A -85,B 0,C 180,E1 16617.496,E2 16617.496} C_VEL
LIN {X 0,Y 466.944,Z 985.884,A -85,B 0,C 180,E1 16616.022,E2 16616.022} C_VEL
LIN {X 0,Y 469.321,Z 966.875,A -85,B 0,C 180,E1 16614.81,E2 16614.81} C_VEL
LIN {X 0,Y 471.536,Z 946.86,A -85,B 0,C 180,E1 16613.767,E2 16613.767} C_VEL
LIN {X 0,Y 473.367,Z 926.285,A -85,B 0,C 180,E1 16612.931,E2 16612.931} C_VEL
LIN {X 0,Y 474.792,Z 905.254,A -85,B 0,C 180,E1 16612.307,E2 16612.307} C_VEL
LIN {X 0,Y 475.717,Z 883.125,A -85,B 0,C 180,E1 16611.856,E2 16611.856} C_VEL
LIN {X 0,Y 480.816,Z 654.206,A -85,B 0,C 180,E1 16608.076,E2 16608.076} C_VEL
LIN {X 0,Y 481.388,Z 623.672,A -85,B 0,C 180,E1 16607.539,E2 16607.539} C_VEL
LIN {X 0,Y 473.928,Z 585.411,A -85,B 0,C 180,E1 16605.792,E2 16605.792} C_VEL
LIN {X 0,Y 474.046,Z 582.386,A -85,B 0,C 180,E1 16605.472,E2 16605.472} C_VEL
LIN {X 0,Y 467.597,Z 566.655,A -85,B 0,C 180,E1 16602.825,E2 16602.825} C_VEL
LIN {X 0,Y 461.451,Z 552.644,A -85,B 0,C 180,E1 16600.218,E2 16600.218} C_VEL
LIN {X 0,Y 459.908,Z 549.42,A -85,B 0,C 180,E1 16599.568,E2 16599.568} C_VEL
LIN {X 0,Y 457.67,Z 549.127,A -85,B 0,C 180,E1 16599.144,E2 16599.144} C_VEL
LIN {X 0,Y 457.672,Z 550.05,A -85,B 0,C 180,E1 16598.896,E2 16598.896} C_VEL
LIN {X 0,Y 462.644,Z 565.347,A -85,B 0,C 180,E1 16597.153,E2 16597.153} C_VEL
LIN {X 0,Y 461.109,Z 608.913,A -85,B 0,C 180,E1 16593.494,E2 16593.494} C_VEL
LIN {X 0,Y 459.606,Z 649.413,A -85,B 0,C 180,E1 16590.096,E2 16590.096} C_VEL
LIN {X 0,Y 457.778,Z 693.562,A -85,B 0,C 180,E1 16586.39,E2 16586.39} C_VEL
LIN {X 0,Y 456.96,Z 716.136,A -85,B 0,C 180,E1 16584.528,E2 16584.528} C_VEL
LIN {X 0,Y 457.884,Z 725.73,A -85,B 0,C 180,E1 16584.298,E2 16584.298} C_VEL
LIN {X 0,Y 455.45,Z 887.347,A -85,B 0,C 180,E1 16581.512,E2 16581.512} C_VEL
LIN {X 0,Y 455.067,Z 904.895,A -85,B 0,C 180,E1 16580.97,E2 16580.97} C_VEL
LIN {X 0,Y 454.47,Z 921.843,A -85,B 0,C 180,E1 16580.207,E2 16580.207} C_VEL
LIN {X 0,Y 453.757,Z 937.973,A -85,B 0,C 180,E1 16579.239,E2 16579.239} C_VEL
LIN {X 0,Y 452.921,Z 953.141,A -85,B 0,C 180,E1 16578.069,E2 16578.069} C_VEL
LIN {X 0,Y 452.069,Z 967.205,A -85,B 0,C 180,E1 16576.71,E2 16576.71} C_VEL
LIN {X 0,Y 451.222,Z 980.268,A -85,B 0,C 180,E1 16575.158,E2 16575.158} C_VEL
LIN {X 0,Y 450.466,Z 991.771,A -85,B 0,C 180,E1 16573.478,E2 16573.478} C_VEL
LIN {X 0,Y 449.83,Z 1001.734,A -85,B 0,C 180,E1 16571.67,E2 16571.67} C_VEL
LIN {X 0,Y 449.31,Z 1010.787,A -85,B 0,C 180,E1 16569.608,E2 16569.608} C_VEL
LIN {X 0,Y 448.971,Z 1017.76,A -85,B 0,C 180,E1 16567.55,E2 16567.55} C_VEL
LIN {X 0,Y 448.764,Z 1023.115,A -85,B 0,C 180,E1 16565.37,E2 16565.37} C_VEL
LIN {X 0,Y 448.68,Z 1026.667,A -85,B 0,C 180,E1 16563.194,E2 16563.194} C_VEL
LIN {X 0,Y 448.678,Z 1028.531,A -85,B 0,C 180,E1 16561.022,E2 16561.022} C_VEL
LIN {X 0,Y 448.712,Z 1028.693,A -85,B 0,C 180,E1 16558.851,E2 16558.851} C_VEL
LIN {X 0,Y 448.776,Z 1027.186,A -85,B 0,C 180,E1 16556.68,E2 16556.68} C_VEL
LIN {X 0,Y 448.931,Z 1023.984,A -85,B 0,C 180,E1 16554.505,E2 16554.505} C_VEL
LIN {X 0,Y 449.188,Z 1019.293,A -85,B 0,C 180,E1 16552.454,E2 16552.454} C_VEL
LIN {X 0,Y 449.577,Z 1012.705,A -85,B 0,C 180,E1 16550.399,E2 16550.399} C_VEL
LIN {X 0,Y 450.124,Z 1004.016,A -85,B 0,C 180,E1 16548.338,E2 16548.338} C_VEL
LIN {X 0,Y 450.774,Z 994.349,A -85,B 0,C 180,E1 16546.533,E2 16546.533} C_VEL
LIN {X 0,Y 451.515,Z 983.046,A -85,B 0,C 180,E1 16544.853,E2 16544.853} C_VEL
LIN {X 0,Y 452.325,Z 970.079,A -85,B 0,C 180,E1 16543.3,E2 16543.3} C_VEL
LIN {X 0,Y 453.06,Z 956.637,A -85,B 0,C 180,E1 16542.003,E2 16542.003} C_VEL
LIN {X 0,Y 453.709,Z 942.225,A -85,B 0,C 180,E1 16540.898,E2 16540.898} C_VEL
LIN {X 0,Y 454.3,Z 925.78,A -85,B 0,C 180,E1 16539.92,E2 16539.92} C_VEL
LIN {X 0,Y 454.727,Z 908.83,A -85,B 0,C 180,E1 16539.178,E2 16539.178} C_VEL
LIN {X 0,Y 454.916,Z 891.183,A -85,B 0,C 180,E1 16538.67,E2 16538.67} C_VEL
LIN {X 0,Y 456.673,Z 763.878,A -85,B 0,C 180,E1 16536.455,E2 16536.455} C_VEL
LIN {X 0,Y 457.484,Z 725.943,A -85,B 0,C 180,E1 16535.74,E2 16535.74} C_VEL
LIN {X 0,Y 458.017,Z 720.732,A -85,B 0,C 180,E1 16535.358,E2 16535.358} C_VEL
LIN {X 0,Y 459.058,Z 680.075,A -85,B 0,C 180,E1 16532.165,E2 16532.165} C_VEL
LIN {X 0,Y 459.639,Z 642.514,A -85,B 0,C 180,E1 16529.329,E2 16529.329} C_VEL
LIN {X 0,Y 459.722,Z 603.959,A -85,B 0,C 180,E1 16526.541,E2 16526.541} C_VEL
LIN {X 0,Y 459.305,Z 562.184,A -85,B 0,C 180,E1 16523.693,E2 16523.693} C_VEL
LIN {X 0,Y 459.01,Z 554.903,A -85,B 0,C 180,E1 16523.2,E2 16523.2} C_VEL
LIN {X 0,Y 457.954,Z 549.308,A -85,B 0,C 180,E1 16522.709,E2 16522.709} C_VEL
LIN {X 0,Y 458.373,Z 548.663,A -85,B 0,C 180,E1 16522.513,E2 16522.513} C_VEL
LIN {X 0,Y 459.826,Z 548.704,A -85,B 0,C 180,E1 16522.259,E2 16522.259} C_VEL
LIN {X 0,Y 461.388,Z 551.44,A -85,B 0,C 180,E1 16521.819,E2 16521.819} C_VEL
LIN {X 0,Y 473.186,Z 567.908,A -85,B 0,C 180,E1 16519.815,E2 16519.815} C_VEL
LIN {X 0,Y 485.813,Z 587.207,A -85,B 0,C 180,E1 16517.817,E2 16517.817} C_VEL
